Fanuc TP program (LS listing): op5_xl_master.ls

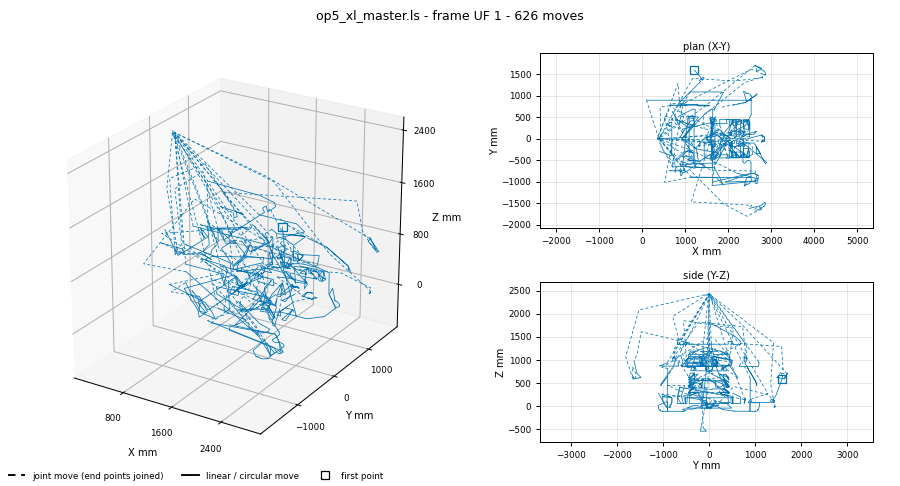
[picture p0: tool path of op5_xl_master.ls in frame UF 1, 626 of 638 moves have a stored position in this frame; points joined in program order, loops and branches not executed]
/PROG  OP5_XL_MASTER
/ATTR
OWNER		= SHIFT;
COMMENT		= "XL Main Prog";
PROG_SIZE	= 81377;
CREATE		= DATE 25-11-17  TIME 10:12:48;
MODIFIED	= DATE 26-02-12  TIME 09:04:14;
FILE_NAME	= OP5_XL_M;
VERSION		= 0;
LINE_COUNT	= 1858;
MEMORY_SIZE	= 81929;
PROTECT		= READ_WRITE;
TCD:  STACK_SIZE	= 0,
      TASK_PRIORITY	= 50,
      TIME_SLICE	= 0,
      BUSY_LAMP_OFF	= 0,
      ABORT_REQUEST	= 0,
      PAUSE_REQUEST	= 0;
DEFAULT_GROUP	= 1,1,*,*,*;
CONTROL_CODE	= 00000000 00000000;
/APPL
  ARC Welding Equipment : 1,*,*,*,*;

MPAS ;
MPAS_NUM_PASSES        : 0;
MPAS_LAST_PASS         : 0;
MPAS_CURRENT_PASS      : 0;
MPAS_STATUS_PASS       : 0;
/MN
   1:  !********** WAR HAMMER ********** ;
   2:  !-           FRAME XL           - ;
   3:  !******** FR500 CELL: C ********* ;
   4:   ;
   5:  CALL HOME    ;
   6:  CALL LOAD_POS    ;
   7:  UFRAME_NUM[GP2]=0 ;
   8:   ;
   9:  !********POSITIONER MOVE******** ;
  10:J P[1] 60% FINE    ;
  11:   ;
  12:L P[2] 1000mm/sec CNT25    ;
  13:   ;
  14:  !FR50X1000 ;
  15:  IF R[15]=1003,CALL TECH_HOLD ;
  16:   ;
  17:L P[3] 800mm/sec FINE
    :  Arc Start[6]    ;
  18:  Weave Sine[6] ;
  19:  Track TAST[6] ;
  20:L P[4] WELD_SPEED FINE
    :  Arc End[6]    ;
  21:  Weave End ;
  22:  Track End ;
  23:   ;
  24:L P[5] 1000mm/sec CNT50    ;
  25:   ;
  26:L P[6] 1000mm/sec CNT50    ;
  27:   ;
  28:   ;
  29:  !FR50X1010 ;
  30:  IF R[15]=1013,CALL TECH_HOLD ;
  31:   ;
  32:L P[7] 800mm/sec FINE
    :  Arc Start[6]    ;
  33:  Weave Sine[6] ;
  34:  Track TAST[6] ;
  35:L P[8] WELD_SPEED FINE
    :  Arc End[6]    ;
  36:  Weave End ;
  37:  Track End ;
  38:   ;
  39:L P[9] 1000mm/sec CNT25    ;
  40:   ;
  41:  !FR50X1020 ;
  42:  IF R[15]=1023,CALL TECH_HOLD ;
  43:   ;
  44:L P[10] 800mm/sec FINE
    :  Arc Start[6]    ;
  45:  Weave Sine[6] ;
  46:  Track TAST[6] ;
  47:L P[11] WELD_SPEED CNT100    ;
  48:L P[12] WELD_SPEED FINE
    :  Arc End[6]    ;
  49:  Weave End ;
  50:  Track End ;
  51:   ;
  52:L P[13] 1000mm/sec CNT25    ;
  53:   ;
  54:J P[14] 50% CNT25    ;
  55:   ;
  56:  !HOME ;
  57:J P[15] 75% CNT25    ;
  58:   ;
  59:  !********POSITIONER MOVE******** ;
  60:J P[16] 75% FINE    ;
  61:   ;
  62:J P[17] 50% CNT100    ;
  63:   ;
  64:J P[18] 50% CNT25    ;
  65:   ;
  66:  !FR50X1030 ;
  67:  IF R[15]=1033,CALL TECH_HOLD ;
  68:   ;
  69:L P[19] 800mm/sec FINE
    :  Arc Start[6]    ;
  70:  Weave Sine[6] ;
  71:  Track TAST[6] ;
  72:L P[20] WELD_SPEED FINE
    :  Arc End[6]    ;
  73:  Weave End ;
  74:  Track End ;
  75:   ;
  76:L P[21] 1000mm/sec CNT25    ;
  77:   ;
  78:J P[22] 50% CNT25    ;
  79:   ;
  80:L P[23] 1000mm/sec CNT25    ;
  81:   ;
  82:  !FR50X1040 ;
  83:  IF R[15]=1043,CALL TECH_HOLD ;
  84:   ;
  85:L P[24] 800mm/sec FINE
    :  Arc Start[6]    ;
  86:  Weave Sine[6] ;
  87:  Track TAST[6] ;
  88:L P[25] WELD_SPEED FINE
    :  Arc End[6]    ;
  89:  Weave End ;
  90:  Track End ;
  91:   ;
  92:L P[26] 960mm/sec CNT25    ;
  93:   ;
  94:J P[27] 50% CNT25    ;
  95:   ;
  96:   ;
  97:L P[28] 1000mm/sec CNT25    ;
  98:   ;
  99:  !FR50X1050 ;
 100:  IF R[15]=1053,CALL TECH_HOLD ;
 101:   ;
 102:L P[29] 800mm/sec FINE
    :  Arc Start[6]    ;
 103:  Weave Sine[6] ;
 104:  Track TAST[6] ;
 105:L P[30] WELD_SPEED CNT100    ;
 106:L P[31] WELD_SPEED FINE
    :  Arc End[6]    ;
 107:  Weave End ;
 108:  Track End ;
 109:   ;
 110:L P[32] 960mm/sec CNT25    ;
 111:   ;
 112:J P[33] 50% CNT25    ;
 113:   ;
 114:L P[34] 1000mm/sec CNT25    ;
 115:   ;
 116:  !FR50X1060 ;
 117:  IF R[15]=1063,CALL TECH_HOLD ;
 118:   ;
 119:L P[35] 800mm/sec FINE
    :  Arc Start[6]    ;
 120:  Weave Sine[6] ;
 121:  Track TAST[6] ;
 122:L P[36] WELD_SPEED CNT100    ;
 123:L P[37] WELD_SPEED FINE
    :  Arc End[6]    ;
 124:  Weave End ;
 125:  Track End ;
 126:   ;
 127:L P[38] 1000mm/sec CNT25    ;
 128:   ;
 129:J P[39] 50% CNT25    ;
 130:   ;
 131:L P[40] 1000mm/sec CNT25    ;
 132:   ;
 133:  !FR50X1070 ;
 134:  IF R[15]=1073,CALL TECH_HOLD ;
 135:   ;
 136:L P[41] 500mm/sec FINE
    :  Arc Start[6]    ;
 137:  Weave Sine[6] ;
 138:  Track TAST[6] ;
 139:L P[42] WELD_SPEED CNT100    ;
 140:L P[43] WELD_SPEED CNT100    ;
 141:L P[44] WELD_SPEED FINE
    :  Arc End[6]    ;
 142:  Weave End ;
 143:  Track End ;
 144:   ;
 145:L P[45] 700mm/sec CNT25    ;
 146:   ;
 147:L P[46] 1000mm/sec CNT50    ;
 148:   ;
 149:  !FR50X1080 ;
 150:  IF R[15]=1083,CALL TECH_HOLD ;
 151:   ;
 152:L P[47] 800mm/sec FINE
    :  Arc Start[6]    ;
 153:  Weave Sine[6] ;
 154:  Track TAST[6] ;
 155:L P[48] WELD_SPEED FINE
    :  Arc End[6]    ;
 156:  Weave End ;
 157:  Track End ;
 158:   ;
 159:L P[49] 1000mm/sec CNT25    ;
 160:   ;
 161:L P[50] 960mm/sec CNT25    ;
 162:   ;
 163:J P[51] 50% CNT25    ;
 164:   ;
 165:L P[52] 1000mm/sec CNT25    ;
 166:   ;
 167:  !FR50X1090 ;
 168:  IF R[15]=1093,CALL TECH_HOLD ;
 169:   ;
 170:L P[53] 800mm/sec FINE
    :  Arc Start[6]    ;
 171:  Weave Sine[6] ;
 172:  Track TAST[6] ;
 173:L P[54] WELD_SPEED CNT100    ;
 174:L P[55] WELD_SPEED CNT100    ;
 175:L P[56] WELD_SPEED FINE
    :  Arc End[6]    ;
 176:  Weave End ;
 177:  Track End ;
 178:   ;
 179:L P[57] 1000mm/sec CNT25    ;
 180:   ;
 181:L P[58] 1000mm/sec CNT50    ;
 182:   ;
 183:  !FR50X1100 ;
 184:  IF R[15]=1103,CALL TECH_HOLD ;
 185:   ;
 186:L P[59] 800mm/sec FINE
    :  Arc Start[6]    ;
 187:  Weave Sine[6] ;
 188:  Track TAST[6] ;
 189:L P[60] WELD_SPEED FINE
    :  Arc End[6]    ;
 190:  Weave End ;
 191:  Track End ;
 192:   ;
 193:L P[61] 1000mm/sec CNT25    ;
 194:   ;
 195:J P[62] 50% CNT25    ;
 196:   ;
 197:L P[63] 1000mm/sec CNT25    ;
 198:   ;
 199:  !FR50X1110 ;
 200:  IF R[15]=1113,CALL TECH_HOLD ;
 201:   ;
 202:L P[64] 800mm/sec FINE
    :  Arc Start[8]    ;
 203:  Weave Sine[8] ;
 204:L P[65] WELD_SPEED CNT100    ;
 205:L P[66] WELD_SPEED FINE
    :  Arc End[8]    ;
 206:  Weave End ;
 207:   ;
 208:L P[67] 800mm/sec CNT25    ;
 209:   ;
 210:J P[68] 50% CNT25    ;
 211:   ;
 212:  !********POSITIONER MOVE******** ;
 213:J P[69] 75% FINE    ;
 214:   ;
 215:  !FR50X1120 ;
 216:  IF R[15]=1123,CALL TECH_HOLD ;
 217:   ;
 218:L P[70] 800mm/sec FINE
    :  Arc Start[8]    ;
 219:  Weave Sine[8] ;
 220:L P[71] WELD_SPEED FINE
    :  Arc End[8]    ;
 221:  Weave End ;
 222:   ;
 223:L P[72] 1000mm/sec CNT25    ;
 224:   ;
 225:J P[73] 50% CNT25    ;
 226:   ;
 227:  !HOME ;
 228:J P[74] 100% FINE    ;
 229:   ;
 230:  !********POSITIONER MOVE******** ;
 231:J P[75] 60% FINE    ;
 232:   ;
 233:J P[76] 50% CNT25    ;
 234:   ;
 235:L P[77] 1000mm/sec CNT25    ;
 236:   ;
 237:L P[78] 500mm/sec CNT25    ;
 238:   ;
 239:  !FR50X1130 ;
 240:  IF R[15]=1133,CALL TECH_HOLD ;
 241:   ;
 242:L P[79] 400mm/sec FINE
    :  Arc Start[6]    ;
 243:  Weave Sine[6] ;
 244:L P[80] WELD_SPEED FINE
    :  Arc End[6]    ;
 245:  Weave End ;
 246:   ;
 247:L P[81] 500mm/sec CNT25    ;
 248:   ;
 249:L P[82] 1000mm/sec CNT25    ;
 250:   ;
 251:J P[83] 40% CNT25    ;
 252:   ;
 253:J P[84] 50% CNT25    ;
 254:   ;
 255:  !HOME ;
 256:J P[85] 100% FINE    ;
 257:   ;
 258:  !********POSITIONER MOVE******** ;
 259:J P[86] 70% FINE    ;
 260:   ;
 261:J P[87] 50% CNT25    ;
 262:   ;
 263:L P[88] 1000mm/sec CNT25    ;
 264:   ;
 265:L P[89] 1000mm/sec CNT25    ;
 266:   ;
 267:  !FR50X1140 ;
 268:  IF R[15]=1143,CALL TECH_HOLD ;
 269:   ;
 270:L P[90] 700mm/sec FINE
    :  Arc Start[6]    ;
 271:  Weave Sine[6] ;
 272:  Track TAST[6] ;
 273:L P[91] WELD_SPEED CNT100    ;
 274:L P[92] WELD_SPEED FINE
    :  Arc End[6]    ;
 275:  Weave End ;
 276:  Track End ;
 277:   ;
 278:L P[93] 1000mm/sec CNT25    ;
 279:   ;
 280:L P[94] 1000mm/sec CNT25    ;
 281:   ;
 282:L P[95] 1000mm/sec CNT25    ;
 283:   ;
 284:J P[96] 50% CNT25    ;
 285:   ;
 286:L P[97] 1000mm/sec CNT25    ;
 287:   ;
 288:  !FR50X1150 ;
 289:  IF R[15]=1153,CALL TECH_HOLD ;
 290:   ;
 291:L P[98] 1000mm/sec FINE
    :  Arc Start[6]    ;
 292:  Weave Sine[6] ;
 293:  Track TAST[6] ;
 294:L P[99] WELD_SPEED CNT100    ;
 295:L P[100] WELD_SPEED FINE
    :  Arc End[6]    ;
 296:  Weave End ;
 297:  Track End ;
 298:   ;
 299:L P[101] 1000mm/sec CNT25    ;
 300:   ;
 301:L P[102] 1000mm/sec CNT25    ;
 302:   ;
 303:  !********POSITIONER MOVE******** ;
 304:J P[103] 75% FINE    ;
 305:   ;
 306:L P[104] 1000mm/sec CNT25    ;
 307:   ;
 308:L P[105] 1000mm/sec CNT25    ;
 309:   ;
 310:  !FR50X1160 ;
 311:  IF R[15]=1163,CALL TECH_HOLD ;
 312:   ;
 313:L P[106] 1000mm/sec FINE
    :  Arc Start[6]    ;
 314:  Weave Sine[6] ;
 315:  Track TAST[6] ;
 316:L P[107] WELD_SPEED FINE
    :  Arc End[6]    ;
 317:  Weave End ;
 318:  Track End ;
 319:   ;
 320:L P[108] 1000mm/sec CNT25    ;
 321:   ;
 322:  !FR50X1170 ;
 323:  IF R[15]=1173,CALL TECH_HOLD ;
 324:   ;
 325:L P[109] 1000mm/sec FINE
    :  Arc Start[6]    ;
 326:  Weave Sine[6] ;
 327:  Track TAST[6] ;
 328:L P[110] WELD_SPEED FINE
    :  Arc End[6]    ;
 329:  Weave End ;
 330:  Track End ;
 331:   ;
 332:L P[111] 1000mm/sec CNT25    ;
 333:   ;
 334:L P[112] 1000mm/sec CNT25    ;
 335:   ;
 336:  !FR50X1180 ;
 337:  IF R[15]=1183,CALL TECH_HOLD ;
 338:   ;
 339:L P[113] 1000mm/sec FINE
    :  Arc Start[6]    ;
 340:  Weave Sine[6] ;
 341:  Track TAST[6] ;
 342:L P[114] WELD_SPEED FINE
    :  Arc End[6]    ;
 343:  Weave End ;
 344:  Track End ;
 345:   ;
 346:L P[115] 1000mm/sec CNT25    ;
 347:   ;
 348:L P[116] 1000mm/sec CNT25    ;
 349:   ;
 350:  !FR50X1190 ;
 351:  IF R[15]=1193,CALL TECH_HOLD ;
 352:   ;
 353:L P[117] 1000mm/sec FINE
    :  Arc Start[6]    ;
 354:  Weave Sine[6] ;
 355:  Track TAST[6] ;
 356:L P[118] WELD_SPEED FINE
    :  Arc End[6]    ;
 357:  Weave End ;
 358:  Track End ;
 359:   ;
 360:L P[119] 1000mm/sec CNT25    ;
 361:   ;
 362:L P[120] 1000mm/sec CNT25    ;
 363:   ;
 364:  !FR50X1200 ;
 365:  IF R[15]=1203,CALL TECH_HOLD ;
 366:   ;
 367:L P[121] 1000mm/sec FINE
    :  Arc Start[6]    ;
 368:  Weave Sine[6] ;
 369:  Track TAST[6] ;
 370:L P[122] WELD_SPEED FINE
    :  Arc End[6]    ;
 371:  Weave End ;
 372:  Track End ;
 373:   ;
 374:L P[123] 1000mm/sec CNT25    ;
 375:   ;
 376:L P[124] 1000mm/sec CNT25    ;
 377:   ;
 378:J P[125] 50% CNT25    ;
 379:   ;
 380:  !********POSITIONER MOVE******** ;
 381:J P[126] 75% FINE    ;
 382:   ;
 383:L P[127] 1000mm/sec CNT25    ;
 384:   ;
 385:  !FR50X1210 ;
 386:  IF R[15]=1213,CALL TECH_HOLD ;
 387:   ;
 388:L P[128] 500mm/sec FINE
    :  Arc Start[6]    ;
 389:  Weave Sine[6] ;
 390:  Track TAST[6] ;
 391:L P[129] WELD_SPEED FINE
    :  Arc End[6]    ;
 392:  Weave End ;
 393:  Track End ;
 394:   ;
 395:L P[130] 500mm/sec CNT25    ;
 396:   ;
 397:L P[131] 1000mm/sec FINE    ;
 398:   ;
 399:J P[132] 50% CNT25    ;
 400:   ;
 401:  !********POSITIONER MOVE******** ;
 402:J P[133] 75% FINE    ;
 403:   ;
 404:J P[134] 50% CNT25    ;
 405:   ;
 406:L P[135] 1000mm/sec CNT25    ;
 407:   ;
 408:  !FR50X1220 ;
 409:  IF R[15]=1223,CALL TECH_HOLD ;
 410:   ;
 411:L P[136] 1000mm/sec FINE
    :  Arc Start[6]    ;
 412:  Weave Sine[6] ;
 413:  Track TAST[6] ;
 414:L P[137] WELD_SPEED FINE
    :  Arc End[6]    ;
 415:  Weave End ;
 416:  Track End ;
 417:   ;
 418:L P[138] 500mm/sec CNT25    ;
 419:   ;
 420:J P[139] 50% CNT25    ;
 421:   ;
 422:J P[140] 50% CNT25    ;
 423:   ;
 424:  !HOME ;
 425:J P[141] 100% FINE    ;
 426:   ;
 427:  !********POSITIONER MOVE******** ;
 428:J P[142] 75% FINE    ;
 429:   ;
 430:  !TORCH CLEAN ;
 431:  CALL T_CLEAN    ;
 432:   ;
 433:   ;
 434:J P[143] 50% CNT25    ;
 435:   ;
 436:L P[144] 960mm/sec CNT25    ;
 437:   ;
 438:  !FR50X1230 ;
 439:  IF R[15]=1233,CALL TECH_HOLD ;
 440:   ;
 441:L P[145] 800mm/sec FINE
    :  Arc Start[6]    ;
 442:  Weave Sine[6] ;
 443:  Track TAST[6] ;
 444:L P[146] WELD_SPEED FINE
    :  Arc End[6]    ;
 445:  Weave End ;
 446:  Track End ;
 447:   ;
 448:L P[147] 960mm/sec CNT25    ;
 449:   ;
 450:J P[148] 50% CNT25    ;
 451:   ;
 452:  !FR50X1240 ;
 453:  IF R[15]=1243,CALL TECH_HOLD ;
 454:   ;
 455:L P[149] 800mm/sec FINE
    :  Arc Start[3]    ;
 456:L P[150] WELD_SPEED CNT100    ;
 457:L P[151] WELD_SPEED FINE
    :  Arc End[3]    ;
 458:   ;
 459:L P[152] 1000mm/sec CNT25    ;
 460:   ;
 461:L P[153] 500mm/sec CNT25    ;
 462:   ;
 463:  //UALM[20] ;
 464:   ;
 465:  !FR50X1250 ;
 466:  IF R[15]=1253,CALL TECH_HOLD ;
 467:   ;
 468:L P[154] 800mm/sec FINE
    :  Arc Start[3]    ;
 469:L P[155] WELD_SPEED CNT100    ;
 470:L P[156] WELD_SPEED FINE
    :  Arc End[3]    ;
 471:   ;
 472:L P[157] 1000mm/sec CNT25    ;
 473:   ;
 474:J P[158] 50% CNT25    ;
 475:   ;
 476:L P[159] 1000mm/sec CNT25    ;
 477:   ;
 478:  !FR50X1260 ;
 479:  IF R[15]=1263,CALL TECH_HOLD ;
 480:   ;
 481:L P[160] 800mm/sec FINE
    :  Arc Start[6]    ;
 482:  Weave Sine[6] ;
 483:  Track TAST[6] ;
 484:L P[161] WELD_SPEED FINE
    :  Arc End[6]    ;
 485:  Track End ;
 486:  Weave End ;
 487:   ;
 488:L P[162] 1000mm/sec CNT25    ;
 489:   ;
 490:L P[163] 1000mm/sec CNT25    ;
 491:   ;
 492:L P[164] 1000mm/sec CNT25    ;
 493:   ;
 494:  !FR50X1270 ;
 495:  IF R[15]=1273,CALL TECH_HOLD ;
 496:   ;
 497:L P[165] 800mm/sec FINE
    :  Arc Start[6]    ;
 498:  Weave Sine[6] ;
 499:  Track TAST[6] ;
 500:L P[166] WELD_SPEED FINE
    :  Arc End[6]    ;
 501:  Weave End ;
 502:  Track End ;
 503:   ;
 504:L P[167] 1000mm/sec CNT25    ;
 505:   ;
 506:J P[168] 50% CNT25    ;
 507:   ;
 508:  !********POSITIONER MOVE******** ;
 509:J P[169] 75% FINE    ;
 510:   ;
 511:L P[170] 1000mm/sec CNT25    ;
 512:   ;
 513:  !FR50X1280 ;
 514:  IF R[15]=1283,CALL TECH_HOLD ;
 515:   ;
 516:L P[171] 1000mm/sec FINE
    :  Arc Start[6]    ;
 517:  Weave Sine[6] ;
 518:  Track TAST[6] ;
 519:L P[172] WELD_SPEED FINE
    :  Arc End[6]    ;
 520:  Weave End ;
 521:  Track End ;
 522:   ;
 523:L P[173] 500mm/sec CNT25    ;
 524:   ;
 525:L P[174] 1000mm/sec CNT25    ;
 526:   ;
 527:L P[175] 1000mm/sec FINE    ;
 528:   ;
 529:  !********POSITIONER MOVE******** ;
 530:J P[176] 75% FINE    ;
 531:   ;
 532:L P[177] 1000mm/sec CNT25    ;
 533:   ;
 534:  !FR50X1290 ;
 535:  IF R[15]=1293,CALL TECH_HOLD ;
 536:   ;
 537:L P[178] 800mm/sec FINE
    :  Arc Start[6]    ;
 538:  Weave Sine[6] ;
 539:  Track TAST[6] ;
 540:L P[179] WELD_SPEED FINE
    :  Arc End[6]    ;
 541:  Weave End ;
 542:  Track End ;
 543:   ;
 544:L P[180] 300mm/sec FINE    ;
 545:   ;
 546:L P[181] 1000mm/sec FINE    ;
 547:   ;
 548:J P[182] 50% CNT25    ;
 549:   ;
 550:  !HOME ;
 551:J P[183] 100% FINE    ;
 552:   ;
 553:  !********POSITIONER MOVE******** ;
 554:J P[184] 75% FINE    ;
 555:   ;
 556:J P[185] 50% CNT25    ;
 557:   ;
 558:   ;
 559:  !FR50X1300 ;
 560:  IF R[15]=1303,CALL TECH_HOLD ;
 561:   ;
 562:   ;
 563:L P[186] 800mm/sec FINE
    :  Arc Start[6]    ;
 564:  Weave Sine[6] ;
 565:  Track TAST[6] ;
 566:L P[187] WELD_SPEED FINE
    :  Arc End[6]    ;
 567:  Weave End ;
 568:  Track End ;
 569:   ;
 570:L P[188] 1000mm/sec CNT25    ;
 571:   ;
 572:L P[189] 1000mm/sec CNT30    ;
 573:   ;
 574:  !FR50X1310 ;
 575:  IF R[15]=1313,CALL TECH_HOLD ;
 576:   ;
 577:L P[190] 800mm/sec FINE
    :  Arc Start[6]    ;
 578:  Weave Sine[6] ;
 579:  Track TAST[6] ;
 580:L P[191] WELD_SPEED FINE
    :  Arc End[6]    ;
 581:  Weave End ;
 582:  Track End ;
 583:   ;
 584:L P[192] 1000mm/sec CNT25    ;
 585:   ;
 586:  !FR50X1320 ;
 587:  IF R[15]=1323,CALL TECH_HOLD ;
 588:   ;
 589:L P[194] 800mm/sec FINE
    :  Arc Start[6]    ;
 590:  Weave Sine[6] ;
 591:  Track TAST[6] ;
 592:L P[195] WELD_SPEED FINE
    :  Arc End[6]    ;
 593:  Weave End ;
 594:  Track End ;
 595:   ;
 596:L P[196] 1000mm/sec CNT25    ;
 597:   ;
 598:  !********POSITIONER MOVE******** ;
 599:J P[197] 100% CNT25    ;
 600:   ;
 601:L P[198] 1000mm/sec CNT25    ;
 602:   ;
 603:  CALL ARC_DISABLE_RH_LS(0) ;
 604:   ;
 605:  //UALM[20] ;
 606:   ;
 607:  !FR50X1330 ;
 608:  IF R[15]=1333,CALL TECH_HOLD ;
 609:   ;
 610:L P[199] 800mm/sec FINE
    :  Arc Start[8]    ;
 611:  Weave Sine[8] ;
 612:L P[200] WELD_SPEED FINE
    :  Arc End[8]    ;
 613:  Weave End ;
 614:   ;
 615:L P[201] 800mm/sec FINE    ;
 616:   ;
 617:L P[202] 1000mm/sec CNT25    ;
 618:   ;
 619:J P[203] 50% CNT25    ;
 620:   ;
 621:  !FR50X1340 ;
 622:  !LENGTH: 57mm ;
 623:  IF R[15]=1343,CALL TECH_HOLD ;
 624:   ;
 625:L P[204] 800mm/sec FINE
    :  Arc Start[8]    ;
 626:  Weave Sine[8] ;
 627:L P[205] WELD_SPEED FINE
    :  Arc End[8]    ;
 628:  Weave End ;
 629:   ;
 630:  CALL ARC_DISABLE_RH_LS(1) ;
 631:   ;
 632:L P[206] 800mm/sec CNT5    ;
 633:   ;
 634:  !********POSITIONER MOVE******** ;
 635:J P[207] 50% CNT25    ;
 636:   ;
 637:J P[208] 50% CNT25    ;
 638:   ;
 639:J P[209] 25% CNT25    ;
 640:   ;
 641:  DO[89:OFF:Inch backward   ]=PULSE,0.8sec ;
 642:   ;
 643:  CALL ARC_LH_DISABLE_LS(0) ;
 644:   ;
 645:  !FR50X1350 ;
 646:  IF R[15]=1353,CALL TECH_HOLD ;
 647:   ;
 648:L P[210] 500mm/sec FINE
    :  Arc Start[8]    ;
 649:  Weave Sine[8] ;
 650:L P[211] WELD_SPEED FINE
    :  Arc End[8]    ;
 651:  Weave End ;
 652:   ;
 653:L P[212] 100mm/sec CNT5    ;
 654:   ;
 655:L P[213] 1000mm/sec CNT25    ;
 656:   ;
 657:J P[214] 100% CNT25    ;
 658:   ;
 659:  !FR50X1360 ;
 660:  !LENGTH: 57mm ;
 661:  IF R[15]=1363,CALL TECH_HOLD ;
 662:   ;
 663:L P[215] 800mm/sec FINE
    :  Arc Start[8]    ;
 664:  Weave Sine[8] ;
 665:L P[216] WELD_SPEED FINE
    :  Arc End[8]    ;
 666:  Weave End ;
 667:   ;
 668:  CALL ARC_LH_DISABLE_LS(1) ;
 669:   ;
 670:L P[217] 100mm/sec CNT25    ;
 671:   ;
 672:J P[218] 100% CNT25    ;
 673:   ;
 674:  !HOME ;
 675:J P[219] 100% FINE    ;
 676:   ;
 677:  !********POSITIONER MOVE******** ;
 678:J P[220] 75% FINE    ;
 679:   ;
 680:J P[221] 50% CNT25    ;
 681:   ;
 682:J P[222] 50% CNT25    ;
 683:   ;
 684:   ;
 685:L P[193] 1000mm/sec CNT25    ;
 686:   ;
 687:  !FR50X1370 ;
 688:  IF R[15]=1373,CALL TECH_HOLD ;
 689:   ;
 690:L P[672] 800mm/sec FINE
    :  Arc Start[6]    ;
 691:  Weave Sine[6] ;
 692:L P[673] WELD_SPEED FINE
    :  Arc End[6]    ;
 693:  Weave End ;
 694:   ;
 695:L P[674] 1000mm/sec CNT25    ;
 696:   ;
 697:J P[675] 50% CNT25    ;
 698:   ;
 699:L P[676] 800mm/sec CNT10    ;
 700:   ;
 701:  !FR50X1380 ;
 702:  IF R[15]=1383,CALL TECH_HOLD ;
 703:   ;
 704:L P[677] 800mm/sec FINE
    :  Arc Start[6]    ;
 705:  Weave Sine[6] ;
 706:L P[678] WELD_SPEED FINE
    :  Arc End[6]    ;
 707:  Weave End ;
 708:   ;
 709:L P[679] 1000mm/sec CNT25    ;
 710:   ;
 711:J P[680] 50% CNT25    ;
 712:   ;
 713:L P[681] 500mm/sec CNT25    ;
 714:   ;
 715:  !FR50X1390 ;
 716:  IF R[15]=1393,CALL TECH_HOLD ;
 717:   ;
 718:L P[682] 800mm/sec FINE
    :  Arc Start[6]    ;
 719:  Weave Sine[6] ;
 720:L P[683] WELD_SPEED FINE
    :  Arc End[6]    ;
 721:  Weave End ;
 722:   ;
 723:L P[684] 500mm/sec CNT25    ;
 724:   ;
 725:J P[685] 50% CNT25    ;
 726:   ;
 727:J P[686] 50% CNT25    ;
 728:   ;
 729:J P[687] 50% CNT30    ;
 730:   ;
 731:   ;
 732:   ;
 733:  !FR50X1400 ;
 734:  IF R[15]=1403,CALL TECH_HOLD ;
 735:   ;
 736:L P[688] 800mm/sec FINE
    :  Arc Start[6]    ;
 737:  Weave Sine[6] ;
 738:  Track TAST[6] ;
 739:L P[689] WELD_SPEED FINE
    :  Arc End[6]    ;
 740:  Weave End ;
 741:  Track End ;
 742:   ;
 743:L P[690] 1000mm/sec CNT25    ;
 744:   ;
 745:L P[691] 1000mm/sec CNT25    ;
 746:   ;
 747:  !FR50X1410 ;
 748:  IF R[15]=1413,CALL TECH_HOLD ;
 749:   ;
 750:L P[692] 800mm/sec FINE
    :  Arc Start[6]    ;
 751:  Weave Sine[6] ;
 752:  Track TAST[6] ;
 753:L P[693] WELD_SPEED FINE
    :  Arc End[6]    ;
 754:  Weave End ;
 755:  Track End ;
 756:   ;
 757:L P[694] 1000mm/sec CNT25    ;
 758:   ;
 759:J P[695] 50% CNT25    ;
 760:   ;
 761:   ;
 762:  !FR50X1420 ;
 763:  IF R[15]=1423,CALL TECH_HOLD ;
 764:   ;
 765:L P[696] 800mm/sec FINE
    :  Arc Start[6]    ;
 766:  Weave Sine[6] ;
 767:  Track TAST[6] ;
 768:L P[697] WELD_SPEED CNT100    ;
 769:C P[698]
    :  P[699] WELD_SPEED FINE
    :  Arc End[6]    ;
 770:  Weave End ;
 771:  Track End ;
 772:   ;
 773:L P[700] 1000mm/sec CNT25    ;
 774:   ;
 775:J P[701] 50% CNT25    ;
 776:   ;
 777:J P[702] 50% CNT25    ;
 778:   ;
 779:   ;
 780:   ;
 781:  !FR50X1430 ;
 782:  IF R[15]=1433,CALL TECH_HOLD ;
 783:   ;
 784:L P[703] 800mm/sec FINE
    :  Arc Start[6]    ;
 785:  Weave Sine[6] ;
 786:  Track TAST[6] ;
 787:L P[704] WELD_SPEED FINE
    :  Arc End[6]    ;
 788:  Track End ;
 789:  Weave End ;
 790:   ;
 791:L P[705] 1000mm/sec CNT25    ;
 792:   ;
 793:L P[706] 1000mm/sec CNT25    ;
 794:   ;
 795:  !FR50X1440 ;
 796:  IF R[15]=1443,CALL TECH_HOLD ;
 797:   ;
 798:L P[707] 800mm/sec FINE
    :  Arc Start[6]    ;
 799:  Weave Sine[6] ;
 800:  Track TAST[6] ;
 801:L P[708] WELD_SPEED FINE
    :  Arc End[6]    ;
 802:  Weave End ;
 803:  Track End ;
 804:   ;
 805:L P[709] 1000mm/sec CNT25    ;
 806:   ;
 807:J P[710] 50% CNT25    ;
 808:   ;
 809:  //UALM[20] ;
 810:  //--eg:TOUCH UP ;
 811:   ;
 812:  !FR50X1450 ;
 813:  IF R[15]=1453,CALL TECH_HOLD ;
 814:   ;
 815:L P[711] 800mm/sec FINE
    :  Arc Start[6]    ;
 816:  Weave Sine[6] ;
 817:  Track TAST[6] ;
 818:L P[712] WELD_SPEED CNT100    ;
 819:C P[713]
    :  P[714] WELD_SPEED FINE
    :  Arc End[6]    ;
 820:  Weave End ;
 821:  Track End ;
 822:   ;
 823:L P[715] 960mm/sec FINE    ;
 824:   ;
 825:J P[716] 50% CNT25    ;
 826:   ;
 827:L P[717] 1000mm/sec CNT25    ;
 828:   ;
 829:  !FR50X1460 ;
 830:  IF R[15]=1463,CALL TECH_HOLD ;
 831:   ;
 832:L P[718] 800mm/sec FINE
    :  Arc Start[6]    ;
 833:  Weave Sine[6] ;
 834:  Track TAST[6] ;
 835:L P[719] WELD_SPEED FINE
    :  Arc End[6]    ;
 836:  Weave End ;
 837:  Track End ;
 838:   ;
 839:L P[720] 1000mm/sec CNT25    ;
 840:   ;
 841:L P[721] 1000mm/sec CNT25    ;
 842:   ;
 843:L P[722] 1000mm/sec CNT25    ;
 844:   ;
 845:L P[723] 1000mm/sec CNT25    ;
 846:   ;
 847:  !FR50X1470 ;
 848:  IF R[15]=1473,CALL TECH_HOLD ;
 849:   ;
 850:L P[724] 200mm/sec FINE
    :  Arc Start[6]    ;
 851:  Weave Sine[6] ;
 852:  Track TAST[6] ;
 853:L P[725] WELD_SPEED FINE
    :  Arc End[6]    ;
 854:  Weave End ;
 855:  Track End ;
 856:   ;
 857:L P[726] 200mm/sec CNT25    ;
 858:   ;
 859:L P[727] 1000mm/sec FINE    ;
 860:   ;
 861:J P[728] 50% FINE    ;
 862:   ;
 863:L P[729] 1000mm/sec CNT25    ;
 864:   ;
 865:  !FR50X1480 ;
 866:  IF R[15]=1483,CALL TECH_HOLD ;
 867:   ;
 868:L P[730] 800mm/sec FINE
    :  Arc Start[6]    ;
 869:  Weave Sine[6] ;
 870:  Track TAST[6] ;
 871:L P[731] WELD_SPEED FINE
    :  Arc End[6]    ;
 872:  Weave End ;
 873:  Track End ;
 874:   ;
 875:L P[732] 1000mm/sec CNT25    ;
 876:   ;
 877:L P[733] 500mm/sec CNT25    ;
 878:   ;
 879:L P[734] 500mm/sec CNT25    ;
 880:   ;
 881:  !FR50X1490 ;
 882:  IF R[15]=1493,CALL TECH_HOLD ;
 883:   ;
 884:L P[735] 300mm/sec FINE
    :  Arc Start[6]    ;
 885:  Weave Sine[6] ;
 886:  Track TAST[6] ;
 887:L P[736] WELD_SPEED FINE
    :  Arc End[6]    ;
 888:  Weave End ;
 889:  Track End ;
 890:   ;
 891:L P[737] 300mm/sec CNT25    ;
 892:   ;
 893:J P[738] 25% FINE    ;
 894:   ;
 895:L P[739] 1000mm/sec CNT25    ;
 896:   ;
 897:  !HOME ;
 898:J P[740] 100% FINE    ;
 899:   ;
 900:  !********POSITIONER MOVE******** ;
 901:J P[741] 75% FINE    ;
 902:   ;
 903:J P[742] 50% CNT40    ;
 904:   ;
 905:L P[743] 1000mm/sec CNT25    ;
 906:   ;
 907:  !FR50X1500 ;
 908:  !LENGTH: 100mm ;
 909:  IF R[15]=1503,CALL TECH_HOLD ;
 910:   ;
 911:L P[744] 800mm/sec FINE
    :  Arc Start[8]    ;
 912:  Weave Sine[8] ;
 913:L P[745] WELD_SPEED FINE
    :  Arc End[8]    ;
 914:  Weave End ;
 915:   ;
 916:L P[746] 1000mm/sec CNT25    ;
 917:   ;
 918:  !FR50X1510 ;
 919:  !LENGTH: 85mm ;
 920:  IF R[15]=1513,CALL TECH_HOLD ;
 921:   ;
 922:L P[747] 800mm/sec FINE
    :  Arc Start[8]    ;
 923:  Weave Sine[8] ;
 924:L P[748] WELD_SPEED FINE
    :  Arc End[8]    ;
 925:  Weave End ;
 926:   ;
 927:L P[749] 1000mm/sec CNT25    ;
 928:   ;
 929:L P[750] 1000mm/sec CNT25    ;
 930:   ;
 931:   ;
 932:  !FR50X1520 ;
 933:  !LENGTH: 100mm - 1 of 2 ;
 934:  IF R[15]=1523,CALL TECH_HOLD ;
 935:   ;
 936:L P[751] 800mm/sec FINE
    :  Arc Start[8]    ;
 937:  Weave Sine[8] ;
 938:L P[752] WELD_SPEED FINE
    :  Arc End[8]    ;
 939:  Weave End ;
 940:   ;
 941:L P[753] 1000mm/sec CNT25    ;
 942:   ;
 943:L P[754] 1000mm/sec CNT100    ;
 944:   ;
 945:   ;
 946:   ;
 947:  !FR50X1530 ;
 948:  !LENGTH: 100mm - 2 of 2 ;
 949:  IF R[15]=1533,CALL TECH_HOLD ;
 950:   ;
 951:L P[755] 800mm/sec FINE
    :  Arc Start[6]    ;
 952:  Weave Sine[6] ;
 953:L P[756] WELD_SPEED FINE
    :  Arc End[6]    ;
 954:  Weave End ;
 955:   ;
 956:L P[757] 1000mm/sec CNT50    ;
 957:   ;
 958:L P[758] 1000mm/sec CNT25    ;
 959:   ;
 960:  !FR50X1540 ;
 961:  !LENGTH: 85mm ;
 962:  IF R[15]=1543,CALL TECH_HOLD ;
 963:   ;
 964:L P[759] 800mm/sec FINE
    :  Arc Start[8]    ;
 965:  Weave Sine[8] ;
 966:L P[760] WELD_SPEED FINE
    :  Arc End[8]    ;
 967:  Weave End ;
 968:   ;
 969:L P[761] 1000mm/sec CNT25    ;
 970:   ;
 971:L P[762] 1000mm/sec CNT25    ;
 972:   ;
 973:J P[763] 50% CNT25    ;
 974:   ;
 975:L P[764] 1000mm/sec CNT25    ;
 976:   ;
 977:  !FR50X1550 ;
 978:  IF R[15]=1553,CALL TECH_HOLD ;
 979:   ;
 980:   ;
 981:L P[765] 800mm/sec FINE
    :  Arc Start[6]    ;
 982:  Weave Sine[6] ;
 983:  Track TAST[6] ;
 984:L P[233] WELD_SPEED CNT100    ;
 985:L P[234] WELD_SPEED CNT100    ;
 986:L P[235] WELD_SPEED CNT100    ;
 987:L P[766] WELD_SPEED FINE
    :  Arc End[6]    ;
 988:  Weave End ;
 989:  Track End ;
 990:   ;
 991:L P[767] 1000mm/sec CNT25    ;
 992:   ;
 993:  !FR50X1560 ;
 994:  IF R[15]=1563,CALL TECH_HOLD ;
 995:   ;
 996:L P[768] 800mm/sec FINE
    :  Arc Start[6]    ;
 997:  Weave Sine[6] ;
 998:  Track TAST[6] ;
 999:C P[769]
    :  P[770] WELD_SPEED FINE
    :  Arc End[6]    ;
1000:  Weave End ;
1001:  Track End ;
1002:   ;
1003:L P[771] 1000mm/sec CNT25    ;
1004:   ;
1005:L P[772] 1000mm/sec CNT25    ;
1006:   ;
1007:  !FR50X1570 ;
1008:  IF R[15]=1573,CALL TECH_HOLD ;
1009:   ;
1010:L P[773] 800mm/sec FINE
    :  Arc Start[6]    ;
1011:  Weave Sine[6] ;
1012:  Track TAST[6] ;
1013:L P[774] WELD_SPEED FINE
    :  Arc End[6]    ;
1014:  Weave End ;
1015:  Track End ;
1016:   ;
1017:L P[775] 1000mm/sec CNT25    ;
1018:   ;
1019:L P[776] 1000mm/sec CNT25    ;
1020:   ;
1021:  !FR50X1580 ;
1022:  IF R[15]=1583,CALL TECH_HOLD ;
1023:   ;
1024:L P[777] 800mm/sec FINE
    :  Arc Start[6]    ;
1025:  Weave Sine[6] ;
1026:  Track TAST[6] ;
1027:L P[778] WELD_SPEED CNT100    ;
1028:L P[779] WELD_SPEED CNT100    ;
1029:L P[780] WELD_SPEED FINE
    :  Arc End[6]    ;
1030:  Weave End ;
1031:  Track End ;
1032:   ;
1033:L P[781] 1000mm/sec CNT25    ;
1034:   ;
1035:L P[782] 1000mm/sec CNT25    ;
1036:   ;
1037:  !FR50X1590 ;
1038:  IF R[15]=1593,CALL TECH_HOLD ;
1039:   ;
1040:L P[783] 800mm/sec FINE
    :  Arc Start[6]    ;
1041:  Weave Sine[6] ;
1042:  Track TAST[6] ;
1043:L P[784] WELD_SPEED FINE
    :  Arc End[6]    ;
1044:  Weave End ;
1045:  Track End ;
1046:   ;
1047:L P[785] 1000mm/sec CNT25    ;
1048:   ;
1049:J P[786] 50% CNT25    ;
1050:   ;
1051:J P[787] 50% CNT25    ;
1052:   ;
1053:  !FR50X1600 ;
1054:  IF R[15]=1603,CALL TECH_HOLD ;
1055:   ;
1056:L P[788] 800mm/sec FINE
    :  Arc Start[6]    ;
1057:  Weave Sine[6] ;
1058:  Track TAST[6] ;
1059:L P[789] WELD_SPEED FINE
    :  Arc End[6]    ;
1060:  Weave End ;
1061:  Track End ;
1062:   ;
1063:L P[790] 1000mm/sec CNT25    ;
1064:   ;
1065:  !FR50X1610 ;
1066:  IF R[15]=1613,CALL TECH_HOLD ;
1067:   ;
1068:L P[791] 800mm/sec FINE
    :  Arc Start[6]    ;
1069:  Weave Sine[6] ;
1070:  Track TAST[6] ;
1071:C P[792]
    :  P[793] WELD_SPEED FINE
    :  Arc End[6]    ;
1072:  Weave End ;
1073:  Track End ;
1074:   ;
1075:L P[794] 1000mm/sec CNT25    ;
1076:   ;
1077:L P[795] 1000mm/sec CNT25    ;
1078:   ;
1079:   ;
1080:  !FR50X1620 ;
1081:  IF R[15]=1623,CALL TECH_HOLD ;
1082:   ;
1083:L P[796] 800mm/sec FINE
    :  Arc Start[6]    ;
1084:  Weave Sine[6] ;
1085:  Track TAST[6] ;
1086:L P[797] WELD_SPEED FINE
    :  Arc End[6]    ;
1087:  Weave End ;
1088:  Track End ;
1089:   ;
1090:L P[798] 1000mm/sec CNT25    ;
1091:   ;
1092:  !FR50X1630 ;
1093:  IF R[15]=1633,CALL TECH_HOLD ;
1094:   ;
1095:L P[799] 800mm/sec FINE
    :  Arc Start[6]    ;
1096:  Weave Sine[6] ;
1097:  Track TAST[6] ;
1098:L P[800] WELD_SPEED CNT100    ;
1099:L P[801] WELD_SPEED CNT100    ;
1100:L P[802] WELD_SPEED FINE
    :  Arc End[6]    ;
1101:  Weave End ;
1102:  Track End ;
1103:   ;
1104:L P[803] 300mm/sec CNT25    ;
1105:   ;
1106:L P[804] 300mm/sec CNT25    ;
1107:   ;
1108:  !FR50X1640 ;
1109:  IF R[15]=1643,CALL TECH_HOLD ;
1110:   ;
1111:L P[805] 800mm/sec FINE
    :  Arc Start[6]    ;
1112:  Weave Sine[6] ;
1113:  Track TAST[6] ;
1114:L P[806] WELD_SPEED FINE
    :  Arc End[6]    ;
1115:  Weave End ;
1116:  Track End ;
1117:   ;
1118:L P[807] 300mm/sec CNT5    ;
1119:   ;
1120:L P[808] 300mm/sec CNT25    ;
1121:   ;
1122:J P[809] 50% CNT25    ;
1123:   ;
1124:  !HOME ;
1125:J P[810] 100% CNT25    ;
1126:   ;
1127:  !TORCH CLEAN ;
1128:  CALL HOME    ;
1129:  CALL T_CLEAN    ;
1130:   ;
1131:   ;
1132:  !********POSITIONER MOVE******** ;
1133:J P[811] 75% CNT25    ;
1134:   ;
1135:J P[812] 50% CNT80    ;
1136:   ;
1137:J P[813] 50% CNT30    ;
1138:   ;
1139:  !CELL ID: C ... ;
1140:   ;
1141:L P[814] 800mm/sec FINE
    :  Arc Start[1]    ;
1142:  WAIT    .15(sec) ;
1143:L P[815] WELD_SPEED FINE
    :  Arc End[1]    ;
1144:   ;
1145:J P[224] 50% CNT50    ;
1146:   ;
1147:L P[225] 800mm/sec FINE
    :  Arc Start[1]    ;
1148:  WAIT    .15(sec) ;
1149:L P[226] WELD_SPEED FINE
    :  Arc End[1]    ;
1150:   ;
1151:J P[227] 50% CNT50    ;
1152:   ;
1153:L P[228] 800mm/sec FINE
    :  Arc Start[1]    ;
1154:  WAIT    .15(sec) ;
1155:L P[229] WELD_SPEED FINE
    :  Arc End[1]    ;
1156:   ;
1157:J P[230] 50% CNT50    ;
1158:J P[816] 50% CNT60    ;
1159:   ;
1160:J P[817] 50% CNT80    ;
1161:   ;
1162:J P[818] 50% CNT60    ;
1163:   ;
1164:J P[819] 50% CNT60    ;
1165:   ;
1166:L P[820] 960mm/sec CNT25    ;
1167:   ;
1168:  !FR50X1650 ;
1169:  IF R[15]=1653,CALL TECH_HOLD ;
1170:   ;
1171:L P[821] 800mm/sec FINE
    :  Arc Start[6]    ;
1172:  Weave Sine[6] ;
1173:  Track TAST[6] ;
1174:L P[822] WELD_SPEED CNT100    ;
1175:C P[823]
    :  P[824] WELD_SPEED CNT100    ;
1176:L P[825] WELD_SPEED CNT100    ;
1177:C P[826]
    :  P[827] WELD_SPEED CNT100    ;
1178:L P[828] WELD_SPEED CNT100    ;
1179:L P[829] WELD_SPEED FINE
    :  Arc End[6]    ;
1180:  Weave End ;
1181:  Track End ;
1182:   ;
1183:L P[830] 1000mm/sec CNT25    ;
1184:   ;
1185:J P[831] 50% CNT25    ;
1186:   ;
1187:L P[832] 1000mm/sec CNT25    ;
1188:   ;
1189:   ;
1190:   ;
1191:  !FR50X1660 ;
1192:  !LENGTH: 40mm ;
1193:  ! ;
1194:  IF R[15]=1663,CALL TECH_HOLD ;
1195:   ;
1196:L P[833] 800mm/sec FINE
    :  Arc Start[6]    ;
1197:  Weave Sine[6] ;
1198:L P[834] WELD_SPEED FINE
    :  Arc End[6]    ;
1199:  Weave End ;
1200:   ;
1201:  CALL LENGTH_CHECK(1660) ;
1202:   ;
1203:L P[835] 1000mm/sec CNT25    ;
1204:   ;
1205:J P[842] 50% CNT10    ;
1206:   ;
1207:J P[843] 50% CNT10    ;
1208:   ;
1209:L P[844] 1000mm/sec CNT25    ;
1210:   ;
1211:  !FR50X1680 ;
1212:  IF R[15]=1683,CALL TECH_HOLD ;
1213:   ;
1214:L P[845] 800mm/sec FINE
    :  Arc Start[6]    ;
1215:  Weave Sine[6] ;
1216:  Track TAST[6] ;
1217:L P[846] WELD_SPEED FINE
    :  Arc End[6]    ;
1218:  Weave End ;
1219:  Track End ;
1220:   ;
1221:L P[847] 1000mm/sec CNT25    ;
1222:   ;
1223:  !********POSITIONER MOVE******** ;
1224:J P[848] 50% FINE    ;
1225:   ;
1226:  !FR50X1690 ;
1227:  IF R[15]=1693,CALL TECH_HOLD ;
1228:   ;
1229:L P[849] 800mm/sec FINE
    :  Arc Start[6]    ;
1230:  Weave Sine[6] ;
1231:  Track TAST[6] ;
1232:L P[850] WELD_SPEED CNT100    ;
1233:L P[851] WELD_SPEED CNT100    ;
1234:L P[852] WELD_SPEED CNT100    ;
1235:C P[853]
    :  P[854] WELD_SPEED CNT100    ;
1236:L P[855] WELD_SPEED CNT100    ;
1237:L P[856] WELD_SPEED CNT100    ;
1238:L P[857] WELD_SPEED CNT100    ;
1239:C P[858]
    :  P[859] WELD_SPEED CNT100    ;
1240:L P[860] WELD_SPEED CNT100    ;
1241:C P[861]
    :  P[862] WELD_SPEED CNT100    ;
1242:C P[863]
    :  P[864] WELD_SPEED CNT100    ;
1243:L P[865] WELD_SPEED FINE
    :  Arc End[6]    ;
1244:  Weave End ;
1245:  Track End ;
1246:   ;
1247:L P[866] 1000mm/sec CNT25    ;
1248:   ;
1249:L P[867] 1000mm/sec CNT25    ;
1250:   ;
1251:  !FR50X1700 ;
1252:  IF R[15]=1703,CALL TECH_HOLD ;
1253:   ;
1254:L P[868] 1000mm/sec FINE
    :  Arc Start[6]    ;
1255:  Weave Sine[6] ;
1256:  Track TAST[6] ;
1257:L P[869] WELD_SPEED CNT100    ;
1258:C P[870]
    :  P[871] WELD_SPEED CNT100    ;
1259:L P[872] WELD_SPEED CNT100    ;
1260:C P[873]
    :  P[874] WELD_SPEED CNT100    ;
1261:L P[875] WELD_SPEED CNT100    ;
1262:C P[876]
    :  P[877] WELD_SPEED CNT100    ;
1263:C P[878]
    :  P[879] WELD_SPEED FINE
    :  Arc End[6]    ;
1264:  Weave End ;
1265:  Track End ;
1266:   ;
1267:L P[880] 1000mm/sec CNT25    ;
1268:   ;
1269:L P[881] 1000mm/sec CNT25    ;
1270:   ;
1271:J P[882] 50% CNT25    ;
1272:   ;
1273:J P[883] 50% CNT25    ;
1274:   ;
1275:  !********POSITIONER MOVE******** ;
1276:J P[884] 75% FINE    ;
1277:   ;
1278:   ;
1279:  !FR50X1710 ;
1280:  IF R[15]=1713,CALL TECH_HOLD ;
1281:   ;
1282:L P[885] 800mm/sec FINE
    :  Arc Start[6]    ;
1283:  Weave Sine[6] ;
1284:  Track TAST[6] ;
1285:L P[236] WELD_SPEED CNT100    ;
1286:C P[886]
    :  P[887] WELD_SPEED CNT100    ;
1287:L P[888] WELD_SPEED CNT100    ;
1288:C P[889]
    :  P[890] WELD_SPEED CNT100    ;
1289:L P[891] WELD_SPEED FINE
    :  Arc End[6]    ;
1290:  Weave End ;
1291:  Track End ;
1292:   ;
1293:L P[892] 1000mm/sec CNT25    ;
1294:   ;
1295:J P[893] 50% CNT25    ;
1296:   ;
1297:  !FR50X1720 ;
1298:  IF R[15]=1723,CALL TECH_HOLD ;
1299:   ;
1300:L P[894] 800mm/sec FINE
    :  Arc Start[6]    ;
1301:  Weave Sine[6] ;
1302:  Track TAST[6] ;
1303:L P[895] WELD_SPEED CNT100    ;
1304:C P[896]
    :  P[897] WELD_SPEED CNT100    ;
1305:C P[898]
    :  P[899] WELD_SPEED CNT100    ;
1306:C P[900]
    :  P[901] WELD_SPEED CNT100    ;
1307:L P[902] WELD_SPEED FINE
    :  Arc End[6]    ;
1308:  Weave End ;
1309:  Track End ;
1310:   ;
1311:L P[903] 1000mm/sec CNT25    ;
1312:   ;
1313:L P[904] 500mm/sec CNT25    ;
1314:   ;
1315:L P[905] 500mm/sec CNT25    ;
1316:   ;
1317:   ;
1318:  !FR50X1730 ;
1319:  IF R[15]=1733,CALL TECH_HOLD ;
1320:   ;
1321:L P[906] 500mm/sec FINE
    :  Arc Start[6]    ;
1322:  Weave Sine[6] ;
1323:  Track TAST[6] ;
1324:L P[907] WELD_SPEED CNT100    ;
1325:L P[908] WELD_SPEED CNT100    ;
1326:L P[909] WELD_SPEED CNT100    ;
1327:L P[910] WELD_SPEED FINE
    :  Arc End[6]    ;
1328:  Weave End ;
1329:  Track End ;
1330:   ;
1331:L P[911] 500mm/sec CNT25    ;
1332:   ;
1333:L P[912] 1000mm/sec CNT25    ;
1334:   ;
1335:  !FR50X1740 ;
1336:  IF R[15]=1743,CALL TECH_HOLD ;
1337:   ;
1338:L P[913] 800mm/sec FINE
    :  Arc Start[6]    ;
1339:  Weave Sine[6] ;
1340:  Track TAST[6] ;
1341:L P[914] WELD_SPEED FINE
    :  Arc End[6]    ;
1342:  Weave End ;
1343:  Track End ;
1344:   ;
1345:L P[915] 960mm/sec CNT40    ;
1346:   ;
1347:J P[916] 50% CNT35    ;
1348:   ;
1349:  !FR50X1750 ;
1350:  IF R[15]=1753,CALL TECH_HOLD ;
1351:   ;
1352:L P[917] 800mm/sec FINE
    :  Arc Start[6]    ;
1353:  Weave Sine[6] ;
1354:L P[918] WELD_SPEED FINE
    :  Arc End[6]    ;
1355:  Weave End ;
1356:   ;
1357:L P[919] 1000mm/sec CNT50    ;
1358:   ;
1359:J P[223] 50% CNT25    ;
1360:   ;
1361:J P[920] 50% CNT25    ;
1362:   ;
1363:  !FR50X1760 ;
1364:  IF R[15]=1763,CALL TECH_HOLD ;
1365:   ;
1366:L P[921] 800mm/sec FINE
    :  Arc Start[6]    ;
1367:  Weave Sine[6] ;
1368:  Track TAST[6] ;
1369:L P[922] WELD_SPEED FINE
    :  Arc End[6]    ;
1370:  Weave End ;
1371:  Track End ;
1372:   ;
1373:L P[923] 500mm/sec CNT25    ;
1374:   ;
1375:J P[924] 50% CNT25    ;
1376:   ;
1377:J P[925] 50% CNT25    ;
1378:   ;
1379:   ;
1380:  !FR50X1770 ;
1381:  IF R[15]=1773,CALL TECH_HOLD ;
1382:   ;
1383:   ;
1384:L P[926] 1000mm/sec FINE
    :  Arc Start[6]    ;
1385:  Weave Sine[6] ;
1386:  Track TAST[6] ;
1387:L P[927] WELD_SPEED FINE
    :  Arc End[6]    ;
1388:  Weave End ;
1389:  Track End ;
1390:   ;
1391:L P[928] 1000mm/sec CNT25    ;
1392:   ;
1393:L P[929] 1000mm/sec CNT25    ;
1394:   ;
1395:J P[930] 50% CNT25    ;
1396:   ;
1397:   ;
1398:  !FR50X1780 ;
1399:  IF R[15]=1783,CALL TECH_HOLD ;
1400:   ;
1401:L P[931] 1000mm/sec FINE
    :  Arc Start[6]    ;
1402:  Weave Sine[6] ;
1403:  Track TAST[6] ;
1404:L P[932] WELD_SPEED FINE
    :  Arc End[6]    ;
1405:  Weave End ;
1406:  Track End ;
1407:   ;
1408:L P[933] 1000mm/sec CNT25    ;
1409:   ;
1410:J P[934] 50% CNT45    ;
1411:   ;
1412:J P[935] 50% CNT40    ;
1413:   ;
1414:  !********POSITIONER MOVE******** ;
1415:J P[936] 80% CNT25    ;
1416:   ;
1417:J P[937] 50% CNT40    ;
1418:   ;
1419:J P[938] 25% CNT15    ;
1420:   ;
1421:L P[231] 450mm/sec CNT25    ;
1422:   ;
1423:  CALL ARC_DISABLE_RH_LS(0) ;
1424:   ;
1425:  !FR50X1790 ;
1426:  IF R[15]=1793,CALL TECH_HOLD ;
1427:   ;
1428:L P[939] 200mm/sec FINE
    :  Arc Start[8]    ;
1429:  Weave Sine[8] ;
1430:L P[940] WELD_SPEED CNT100    ;
1431:C P[941]
    :  P[942] WELD_SPEED CNT100    ;
1432:L P[943] WELD_SPEED FINE
    :  Arc End[8]    ;
1433:  Weave End ;
1434:   ;
1435:L P[944] 200mm/sec CNT15    ;
1436:   ;
1437:J P[945] 50% CNT25    ;
1438:   ;
1439:  !FR50X1800 ;
1440:  IF R[15]=1803,CALL TECH_HOLD ;
1441:   ;
1442:L P[946] 300mm/sec FINE
    :  Arc Start[8]    ;
1443:  Weave Sine[8] ;
1444:L P[947] WELD_SPEED FINE
    :  Arc End[8]    ;
1445:  Weave End ;
1446:   ;
1447:  CALL ARC_DISABLE_RH_LS(1) ;
1448:   ;
1449:L P[948] 300mm/sec CNT25    ;
1450:   ;
1451:J P[949] 50% CNT25    ;
1452:   ;
1453:  !HOME ;
1454:J P[950] 100% CNT25    ;
1455:   ;
1456:  !TORCH CLEAN ;
1457:  CALL HOME    ;
1458:  CALL T_CLEAN    ;
1459:   ;
1460:  !********POSITIONER MOVE******** ;
1461:J P[951] 75% FINE    ;
1462:   ;
1463:J P[952] 50% CNT25    ;
1464:   ;
1465:L P[953] 1000mm/sec CNT25    ;
1466:   ;
1467:  !FR50X1810 ;
1468:  IF R[15]=1813,CALL TECH_HOLD ;
1469:   ;
1470:L P[954] 800mm/sec FINE
    :  Arc Start[6]    ;
1471:  Weave Sine[6] ;
1472:  Track TAST[6] ;
1473:L P[955] WELD_SPEED FINE
    :  Arc End[6]    ;
1474:  Weave End ;
1475:  Track End ;
1476:   ;
1477:L P[956] 300mm/sec CNT25    ;
1478:   ;
1479:L P[957] 1000mm/sec CNT25    ;
1480:   ;
1481:J P[958] 50% CNT25    ;
1482:   ;
1483:J P[959] 50% CNT25    ;
1484:   ;
1485:L P[960] 1000mm/sec CNT25    ;
1486:   ;
1487:  !FR50X1820 ;
1488:  IF R[15]=1823,CALL TECH_HOLD ;
1489:   ;
1490:L P[961] 1000mm/sec FINE
    :  Arc Start[6]    ;
1491:  Weave Sine[6] ;
1492:  Track TAST[6] ;
1493:C P[962]
    :  P[963] WELD_SPEED CNT100    ;
1494:L P[964] WELD_SPEED FINE
    :  Arc End[6]    ;
1495:  Weave End ;
1496:  Track End ;
1497:   ;
1498:L P[965] 300mm/sec CNT25    ;
1499:   ;
1500:L P[966] 1000mm/sec CNT25    ;
1501:   ;
1502:  !HOME ;
1503:J P[967] 100% CNT25    ;
1504:   ;
1505:  !********POSITIONER MOVE******** ;
1506:J P[968] 75% FINE    ;
1507:   ;
1508:L P[969] 1000mm/sec CNT25    ;
1509:   ;
1510:  !FR50X1830 ;
1511:  IF R[15]=1833,CALL TECH_HOLD ;
1512:   ;
1513:L P[970] 1000mm/sec FINE
    :  Arc Start[6]    ;
1514:  Weave Sine[6] ;
1515:  Track TAST[6] ;
1516:C P[971]
    :  P[972] WELD_SPEED CNT100    ;
1517:L P[973] WELD_SPEED FINE
    :  Arc End[6]    ;
1518:  Weave End ;
1519:  Track End ;
1520:   ;
1521:L P[974] 300mm/sec CNT25    ;
1522:   ;
1523:L P[975] 1000mm/sec CNT25    ;
1524:   ;
1525:  !HOME ;
1526:J P[976] 100% FINE    ;
1527:   ;
1528:  !********POSITIONER MOVE******** ;
1529:J P[977] 75% CNT25    ;
1530:   ;
1531:J P[978] 50% CNT25    ;
1532:   ;
1533:L P[979] 1000mm/sec CNT25    ;
1534:   ;
1535:  //UALM[20] ;
1536:  !DOUBLE CHECK ;
1537:   ;
1538:   ;
1539:  !FR50X1840 ;
1540:  !LENGTH: 40mm ;
1541:   ;
1542:  IF R[15]=1843,CALL TECH_HOLD ;
1543:   ;
1544:L P[980] 800mm/sec FINE
    :  Arc Start[6]    ;
1545:  Weave Sine[6] ;
1546:L P[981] WELD_SPEED FINE
    :  Arc End[6]    ;
1547:  Weave End ;
1548:   ;
1549:  CALL LENGTH_CHECK(1840) ;
1550:   ;
1551:L P[982] 1000mm/sec CNT25    ;
1552:   ;
1553:L P[983] 1000mm/sec CNT25    ;
1554:   ;
1555:J P[984] 50% CNT25    ;
1556:   ;
1557:L P[985] 1000mm/sec CNT25    ;
1558:   ;
1559:  !FR50X1850 ;
1560:  IF R[15]=1853,CALL TECH_HOLD ;
1561:   ;
1562:L P[986] 800mm/sec FINE
    :  Arc Start[6]    ;
1563:  Weave Sine[6] ;
1564:L P[987] WELD_SPEED CNT100    ;
1565:C P[988]
    :  P[989] WELD_SPEED FINE
    :  Arc End[6]    ;
1566:  Weave End ;
1567:   ;
1568:L P[990] 500mm/sec CNT25    ;
1569:   ;
1570:L P[991] 1000mm/sec CNT25    ;
1571:   ;
1572:J P[992] 50% CNT25    ;
1573:   ;
1574:L P[993] 1000mm/sec CNT25    ;
1575:   ;
1576:L P[994] 500mm/sec CNT25    ;
1577:   ;
1578:  !FR50X1860 ;
1579:  IF R[15]=1863,CALL TECH_HOLD ;
1580:   ;
1581:L P[995] 800mm/sec FINE
    :  Arc Start[6]    ;
1582:  Weave Sine[6] ;
1583:L P[996] WELD_SPEED CNT100    ;
1584:C P[997]
    :  P[998] WELD_SPEED FINE
    :  Arc End[6]    ;
1585:  Weave End ;
1586:   ;
1587:L P[999] 300mm/sec CNT5    ;
1588:   ;
1589:L P[1000] 500mm/sec CNT5    ;
1590:   ;
1591:L P[1001] 1000mm/sec CNT25    ;
1592:   ;
1593:J P[1002] 50% CNT25    ;
1594:   ;
1595:L P[1003] 1000mm/sec CNT25    ;
1596:   ;
1597:  !FR50X1870 ;
1598:  IF R[15]=1873,CALL TECH_HOLD ;
1599:   ;
1600:L P[1004] 800mm/sec FINE
    :  Arc Start[6]    ;
1601:  Weave Sine[6] ;
1602:  Track TAST[6] ;
1603:C P[1005]
    :  P[1006] WELD_SPEED CNT100    ;
1604:L P[1007] WELD_SPEED CNT100    ;
1605:C P[1008]
    :  P[1009] WELD_SPEED CNT100    ;
1606:L P[1010] WELD_SPEED CNT100    ;
1607:C P[1011]
    :  P[1012] WELD_SPEED CNT100    ;
1608:L P[1013] WELD_SPEED FINE
    :  Arc End[6]    ;
1609:  Weave End ;
1610:  Track End ;
1611:   ;
1612:L P[1014] 1000mm/sec CNT50    ;
1613:   ;
1614:J P[1015] 50% CNT10    ;
1615:   ;
1616:L P[1016] 1000mm/sec CNT25    ;
1617:   ;
1618:  !FR50X1880 ;
1619:  IF R[15]=1883,CALL TECH_HOLD ;
1620:   ;
1621:L P[1017] 800mm/sec FINE
    :  Arc Start[6]    ;
1622:  Weave Sine[6] ;
1623:  Track TAST[6] ;
1624:L P[1018] WELD_SPEED FINE
    :  Arc End[6]    ;
1625:  Weave End ;
1626:  Track End ;
1627:   ;
1628:L P[1019] 1000mm/sec CNT25    ;
1629:   ;
1630:  !********POSITIONER MOVE******** ;
1631:J P[1020] 75% FINE    ;
1632:   ;
1633:  !FR50X1890 ;
1634:  IF R[15]=1893,CALL TECH_HOLD ;
1635:   ;
1636:L P[1021] 800mm/sec FINE
    :  Arc Start[6]    ;
1637:  Weave Sine[6] ;
1638:  Track TAST[6] ;
1639:L P[1022] WELD_SPEED CNT100    ;
1640:C P[1023]
    :  P[1024] WELD_SPEED CNT100    ;
1641:L P[1025] WELD_SPEED CNT100    ;
1642:C P[1026]
    :  P[1027] WELD_SPEED CNT100    ;
1643:L P[1028] WELD_SPEED CNT100    ;
1644:C P[1029]
    :  P[1030] WELD_SPEED CNT100    ;
1645:L P[1031] WELD_SPEED FINE
    :  Arc End[6]    ;
1646:  Weave End ;
1647:  Track End ;
1648:   ;
1649:L P[1032] 1000mm/sec CNT25    ;
1650:   ;
1651:L P[1033] 1000mm/sec CNT25    ;
1652:   ;
1653:  !FR50X1900 ;
1654:  IF R[15]=1903,CALL TECH_HOLD ;
1655:   ;
1656:L P[1034] 800mm/sec FINE
    :  Arc Start[6]    ;
1657:  Weave Sine[6] ;
1658:  Track TAST[6] ;
1659:L P[1035] WELD_SPEED CNT100    ;
1660:C P[1036]
    :  P[1037] WELD_SPEED CNT100    ;
1661:L P[1038] WELD_SPEED CNT100    ;
1662:C P[1039]
    :  P[1040] WELD_SPEED CNT100    ;
1663:L P[1041] WELD_SPEED CNT100    ;
1664:C P[1042]
    :  P[1043] WELD_SPEED CNT100    ;
1665:C P[1044]
    :  P[1045] WELD_SPEED FINE
    :  Arc End[6]    ;
1666:  Weave End ;
1667:  Track End ;
1668:   ;
1669:L P[1046] 1000mm/sec CNT25    ;
1670:   ;
1671:L P[1047] 1000mm/sec CNT25    ;
1672:   ;
1673:L P[1048] 1000mm/sec CNT25    ;
1674:   ;
1675:L P[1049] 1000mm/sec CNT25    ;
1676:   ;
1677:  !HOME ;
1678:J P[1050] 100% FINE    ;
1679:   ;
1680:  !********POSITIONER MOVE******** ;
1681:J P[1051] 50% CNT25    ;
1682:   ;
1683:  !FR50X1910 ;
1684:  IF R[15]=1913,CALL TECH_HOLD ;
1685:   ;
1686:L P[1052] 780mm/sec FINE
    :  Arc Start[6]    ;
1687:  Weave Sine[6] ;
1688:  Track TAST[6] ;
1689:L P[1053] WELD_SPEED CNT100    ;
1690:C P[1054]
    :  P[1055] WELD_SPEED CNT100    ;
1691:L P[1056] WELD_SPEED CNT100    ;
1692:C P[1057]
    :  P[1058] WELD_SPEED FINE
    :  Arc End[6]    ;
1693:  Weave End ;
1694:  Track End ;
1695:   ;
1696:L P[1059] 1000mm/sec CNT25    ;
1697:   ;
1698:J P[1060] 50% CNT25    ;
1699:   ;
1700:  !FR50X1920 ;
1701:  IF R[15]=1923,CALL TECH_HOLD ;
1702:   ;
1703:L P[1061] 800mm/sec FINE
    :  Arc Start[6]    ;
1704:  Weave Sine[6] ;
1705:  Track TAST[6] ;
1706:L P[1062] WELD_SPEED CNT100    ;
1707:C P[1063]
    :  P[1064] WELD_SPEED CNT100    ;
1708:C P[1065]
    :  P[1066] WELD_SPEED CNT100    ;
1709:C P[1067]
    :  P[1068] WELD_SPEED CNT100    ;
1710:L P[1069] WELD_SPEED FINE
    :  Arc End[6]    ;
1711:  Weave End ;
1712:  Track End ;
1713:   ;
1714:L P[1070] 1000mm/sec CNT25    ;
1715:   ;
1716:L P[1071] 1000mm/sec CNT25    ;
1717:   ;
1718:  !FR50X1930 ;
1719:  IF R[15]=1933,CALL TECH_HOLD ;
1720:   ;
1721:L P[1072] 800mm/sec FINE
    :  Arc Start[6]    ;
1722:  Weave Sine[6] ;
1723:  Track TAST[6] ;
1724:L P[1073] WELD_SPEED FINE
    :  Arc End[6]    ;
1725:  Weave End ;
1726:  Track End ;
1727:   ;
1728:L P[1074] 1000mm/sec CNT25    ;
1729:   ;
1730:L P[1075] 1000mm/sec CNT50    ;
1731:   ;
1732:  !FR50X1940 ;
1733:  IF R[15]=1943,CALL TECH_HOLD ;
1734:   ;
1735:L P[1076] 800mm/sec FINE
    :  Arc Start[6]    ;
1736:  Weave Sine[6] ;
1737:L P[1077] WELD_SPEED FINE
    :  Arc End[6]    ;
1738:  Weave End ;
1739:   ;
1740:L P[1078] 1000mm/sec CNT50    ;
1741:   ;
1742:J P[1079] 50% CNT25    ;
1743:   ;
1744:  !FR50X1950 ;
1745:  IF R[15]=1953,CALL TECH_HOLD ;
1746:   ;
1747:L P[1080] 800mm/sec FINE
    :  Arc Start[6]    ;
1748:  Weave Sine[6] ;
1749:  Track TAST[6] ;
1750:L P[1081] WELD_SPEED FINE
    :  Arc End[6]    ;
1751:  Weave End ;
1752:  Track End ;
1753:   ;
1754:L P[1082] 1000mm/sec CNT25    ;
1755:   ;
1756:J P[1083] 50% CNT25    ;
1757:   ;
1758:J P[1084] 50% CNT25    ;
1759:   ;
1760:  !FR50X1960 ;
1761:  IF R[15]=1963,CALL TECH_HOLD ;
1762:   ;
1763:L P[1085] 800mm/sec FINE
    :  Arc Start[6]    ;
1764:  Weave Sine[6] ;
1765:L P[1086] WELD_SPEED FINE
    :  Arc End[6]    ;
1766:  Weave End ;
1767:   ;
1768:L P[1087] 1000mm/sec CNT100    ;
1769:   ;
1770:J P[1088] 50% CNT30    ;
1771:   ;
1772:  !FR50X1970 ;
1773:  IF R[15]=1973,CALL TECH_HOLD ;
1774:   ;
1775:L P[1089] 780mm/sec FINE
    :  Arc Start[6]    ;
1776:  Weave Sine[6] ;
1777:L P[1090] WELD_SPEED FINE
    :  Arc End[6]    ;
1778:  Weave End ;
1779:   ;
1780:L P[1091] 1000mm/sec CNT75    ;
1781:   ;
1782:J P[1092] 50% CNT40    ;
1783:   ;
1784:  !********POSITIONER MOVE******** ;
1785:J P[1093] 75% CNT25    ;
1786:   ;
1787:J P[1094] 50% CNT25    ;
1788:   ;
1789:J P[1095] 50% CNT30    ;
1790:   ;
1791:L P[1096] 1000mm/sec CNT70    ;
1792:   ;
1793:L P[232] 500mm/sec CNT50    ;
1794:   ;
1795:  CALL ARC_LH_DISABLE_LS(0) ;
1796:   ;
1797:  !FR50X1980 ;
1798:  IF R[15]=1983,CALL TECH_HOLD ;
1799:   ;
1800:L P[1097] 200mm/sec FINE
    :  Arc Start[8]    ;
1801:  Weave Sine[8] ;
1802:L P[1098] WELD_SPEED CNT100    ;
1803:C P[1099]
    :  P[1100] WELD_SPEED CNT100    ;
1804:L P[1101] WELD_SPEED FINE
    :  Arc End[8]    ;
1805:  Weave End ;
1806:   ;
1807:J P[1102] 50% CNT40    ;
1808:   ;
1809:J P[1103] 50% CNT70    ;
1810:   ;
1811:J P[1104] 50% CNT35    ;
1812:   ;
1813:  !FR50X1990 ;
1814:  IF R[15]=1993,CALL TECH_HOLD ;
1815:   ;
1816:L P[1105] 800mm/sec FINE
    :  Arc Start[8]    ;
1817:  Weave Sine[8] ;
1818:L P[1106] WELD_SPEED FINE
    :  Arc End[8]    ;
1819:  Weave End ;
1820:   ;
1821:  CALL ARC_LH_DISABLE_LS(1) ;
1822:   ;
1823:J P[1107] 25% CNT40    ;
1824:   ;
1825:J P[1108] 50% CNT25    ;
1826:   ;
1827:J P[1109] 50% CNT50    ;
1828:   ;
1829:  !HOME ;
1830:J P[1110] 100% CNT25    ;
1831:   ;
1832:  !********POSITIONER MOVE******** ;
1833:J P[1111] 75% FINE    ;
1834:   ;
1835:J P[1112] 50% CNT25    ;
1836:   ;
1837:L P[1113] 1000mm/sec CNT25    ;
1838:   ;
1839:L P[1114] 500mm/sec CNT25    ;
1840:   ;
1841:  !FR50X2000 ;
1842:  IF R[15]=2003,CALL TECH_HOLD ;
1843:   ;
1844:L P[1115] 800mm/sec FINE
    :  Arc Start[6]    ;
1845:  Weave Sine[6] ;
1846:L P[1116] WELD_SPEED FINE
    :  Arc End[6]    ;
1847:  Weave End ;
1848:   ;
1849:L P[1117] 500mm/sec CNT25    ;
1850:   ;
1851:L P[1118] 1000mm/sec CNT25    ;
1852:   ;
1853:J P[1119] 50% CNT25    ;
1854:   ;
1855:   ;
1856:  CALL HOME    ;
1857:  CALL LOAD_POS    ;
1858:   ;
/POS
P[1]{
   GP1:
	UF : 1, UT : 1,		CONFIG : 'N U T, 0, 0, 0',
	X =  1214.464  mm,	Y =  1589.090  mm,	Z =   593.946  mm,
	W =      .000 deg,	P =    44.876 deg,	R =   135.007 deg
   GP2:
	UF : 0, UT : 1,
	J1=     0.000 deg,	J2=    45.000 deg
};
P[2]{
   GP1:
	UF : 1, UT : 1,		CONFIG : 'N U T, 0, 0, 0',
	X =  1343.971  mm,	Y =  1452.300  mm,	Z =   232.946  mm,
	W =      .000 deg,	P =    44.876 deg,	R =   135.007 deg
   GP2:
	UF : 0, UT : 1,
	J1=     0.000 deg,	J2=    45.000 deg
};
P[3]{
   GP1:
	UF : 1, UT : 1,		CONFIG : 'N U T, 0, 0, 0',
	X =  1390.272  mm,	Y =  1354.500  mm,	Z =    79.223  mm,
	W =      .004 deg,	P =    44.873 deg,	R =   131.158 deg
   GP2:
	UF : 0, UT : 1,
	J1=     0.000 deg,	J2=    45.000 deg
};
P[4]{
   GP1:
	UF : 1, UT : 1,		CONFIG : 'N U T, 0, 0, 0',
	X =  1442.813  mm,	Y =  1410.035  mm,	Z =    81.944  mm,
	W =     -.001 deg,	P =    44.845 deg,	R =   152.019 deg
   GP2:
	UF : 0, UT : 1,
	J1=     0.000 deg,	J2=    45.000 deg
};
P[5]{
   GP1:
	UF : 1, UT : 1,		CONFIG : 'N U T, 0, 0, 0',
	X =  1406.269  mm,	Y =  1426.258  mm,	Z =   124.762  mm,
	W =     -.002 deg,	P =    44.845 deg,	R =   152.019 deg
   GP2:
	UF : 0, UT : 1,
	J1=     0.000 deg,	J2=    45.000 deg
};
P[6]{
   GP1:
	UF : 1, UT : 1,		CONFIG : 'N U T, 0, 0, 0',
	X =  1327.201  mm,	Y =  1350.025  mm,	Z =   146.947  mm,
	W =     -.000 deg,	P =    44.876 deg,	R =   131.152 deg
   GP2:
	UF : 0, UT : 1,
	J1=     0.000 deg,	J2=    45.000 deg
};
P[7]{
   GP1:
	UF : 1, UT : 1,		CONFIG : 'N U T, 0, 0, 0',
	X =  1360.318  mm,	Y =  1328.105  mm,	Z =    81.017  mm,
	W =      .000 deg,	P =    44.876 deg,	R =   131.152 deg
   GP2:
	UF : 0, UT : 1,
	J1=     0.000 deg,	J2=    45.000 deg
};
P[8]{
   GP1:
	UF : 1, UT : 1,		CONFIG : 'N U T, 0, 0, 0',
	X =   968.269  mm,	Y =   941.123  mm,	Z =    79.601  mm,
	W =      .000 deg,	P =    44.876 deg,	R =   127.977 deg
   GP2:
	UF : 0, UT : 1,
	J1=     0.000 deg,	J2=    45.000 deg
};
P[9]{
   GP1:
	UF : 1, UT : 1,		CONFIG : 'N U T, 0, 0, 0',
	X =   922.593  mm,	Y =   918.484  mm,	Z =   118.901  mm,
	W =     -.000 deg,	P =    44.876 deg,	R =   129.337 deg
   GP2:
	UF : 0, UT : 1,
	J1=     0.000 deg,	J2=    45.000 deg
};
P[10]{
   GP1:
	UF : 1, UT : 1,		CONFIG : 'N U T, 0, 0, 0',
	X =   932.883  mm,	Y =   905.922  mm,	Z =    80.529  mm,
	W =      .005 deg,	P =    44.838 deg,	R =   129.334 deg
   GP2:
	UF : 0, UT : 1,
	J1=     0.000 deg,	J2=    45.000 deg
};
P[11]{
   GP1:
	UF : 1, UT : 1,		CONFIG : 'N U T, 0, 0, 0',
	X =   885.701  mm,	Y =   855.031  mm,	Z =    77.818  mm,
	W =      .000 deg,	P =    44.876 deg,	R =   129.337 deg
   GP2:
	UF : 0, UT : 1,
	J1=     0.000 deg,	J2=    45.000 deg
};
P[12]{
   GP1:
	UF : 1, UT : 1,		CONFIG : 'N U T, 0, 0, 0',
	X =   879.676  mm,	Y =   853.017  mm,	Z =    79.876  mm,
	W =      .003 deg,	P =    44.796 deg,	R =   114.722 deg
   GP2:
	UF : 0, UT : 1,
	J1=     0.000 deg,	J2=    45.000 deg
};
P[13]{
   GP1:
	UF : 1, UT : 1,		CONFIG : 'N U T, 0, 0, 0',
	X =   863.490  mm,	Y =   904.621  mm,	Z =   146.286  mm,
	W =      .000 deg,	P =    44.876 deg,	R =   112.101 deg
   GP2:
	UF : 0, UT : 1,
	J1=     0.000 deg,	J2=    45.000 deg
};
P[14]{
   GP1:
	UF : 1, UT : 1,		CONFIG : 'N U T, 0, 0, 0',
	X =   831.040  mm,	Y =  1277.928  mm,	Z =   275.925  mm,
	W =      .000 deg,	P =    44.876 deg,	R =   112.101 deg
   GP2:
	UF : 0, UT : 1,
	J1=     0.000 deg,	J2=    45.000 deg
};
P[15]{
   GP1:
	UF : 1, UT : 1,		CONFIG : 'N U B, 0, 0, 0',
	X =   353.784  mm,	Y =     3.997  mm,	Z =  2425.735  mm,
	W =     -.021 deg,	P =   -39.773 deg,	R =      .020 deg
   GP2:
	UF : 1, UT : 1,
	J1=     0.000 deg,	J2=    45.000 deg
};
P[16]{
   GP1:
	UF : 1, UT : 1,
	J1=    -2.565 deg,	J2=   -47.918 deg,	J3=    37.877 deg,
	J4=   -63.535 deg,	J5=   -19.106 deg,	J6=    56.044 deg
   GP2:
	UF : 0, UT : 1,
	J1=     0.000 deg,	J2=   180.000 deg
};
P[17]{
   GP1:
	UF : 1, UT : 1,		CONFIG : 'N U T, 0, 0, 0',
	X =  2036.678  mm,	Y =   133.789  mm,	Z =  1445.358  mm,
	W =   -25.929 deg,	P =   -45.424 deg,	R =    36.423 deg
   GP2:
	UF : 0, UT : 1,
	J1=     0.000 deg,	J2=   180.000 deg
};
P[18]{
   GP1:
	UF : 1, UT : 1,		CONFIG : 'N U T, 0, 0, 0',
	X =  2233.304  mm,	Y =   372.944  mm,	Z =  1162.580  mm,
	W =   -27.414 deg,	P =   -38.078 deg,	R =    43.574 deg
   GP2:
	UF : 0, UT : 1,
	J1=     0.000 deg,	J2=   180.000 deg
};
P[19]{
   GP1:
	UF : 1, UT : 1,		CONFIG : 'N U T, 0, 0, 0',
	X =  2281.974  mm,	Y =   431.829  mm,	Z =  1116.684  mm,
	W =   -41.778 deg,	P =   -28.391 deg,	R =    61.958 deg
   GP2:
	UF : 0, UT : 1,
	J1=      .000 deg,	J2=   180.000 deg
};
P[20]{
   GP1:
	UF : 1, UT : 1,		CONFIG : 'N U T, 0, 0, 0',
	X =  2287.244  mm,	Y =    94.810  mm,	Z =  1116.986  mm,
	W =   -31.951 deg,	P =   -39.356 deg,	R =    44.493 deg
   GP2:
	UF : 0, UT : 1,
	J1=      .000 deg,	J2=   180.000 deg
};
P[21]{
   GP1:
	UF : 1, UT : 1,		CONFIG : 'N U T, 0, 0, 0',
	X =  2124.976  mm,	Y =    85.873  mm,	Z =  1194.632  mm,
	W =   -28.024 deg,	P =   -38.698 deg,	R =    43.953 deg
   GP2:
	UF : 0, UT : 1,
	J1=     0.000 deg,	J2=   180.000 deg
};
P[22]{
   GP1:
	UF : 1, UT : 1,		CONFIG : 'N U T, 0, 0, 0',
	X =  2124.976  mm,	Y =  -285.127  mm,	Z =  1194.632  mm,
	W =    36.159 deg,	P =   -31.426 deg,	R =   -50.949 deg
   GP2:
	UF : 0, UT : 1,
	J1=     0.000 deg,	J2=   180.000 deg
};
P[23]{
   GP1:
	UF : 1, UT : 1,		CONFIG : 'N U T, 0, 0, 0',
	X =  2228.976  mm,	Y =  -404.127  mm,	Z =  1194.631  mm,
	W =    36.159 deg,	P =   -31.426 deg,	R =   -50.949 deg
   GP2:
	UF : 0, UT : 1,
	J1=     0.000 deg,	J2=   180.000 deg
};
P[24]{
   GP1:
	UF : 1, UT : 1,		CONFIG : 'N U T, 0, 0, 0',
	X =  2286.216  mm,	Y =  -430.685  mm,	Z =  1116.208  mm,
	W =    43.325 deg,	P =   -25.600 deg,	R =   -65.383 deg
   GP2:
	UF : 0, UT : 1,
	J1=      .000 deg,	J2=   180.000 deg
};
P[25]{
   GP1:
	UF : 1, UT : 1,		CONFIG : 'N U T, 0, 0, 0',
	X =  2285.704  mm,	Y =   -96.057  mm,	Z =  1118.736  mm,
	W =    36.109 deg,	P =   -35.685 deg,	R =   -49.851 deg
   GP2:
	UF : 0, UT : 1,
	J1=      .000 deg,	J2=   180.000 deg
};
P[26]{
   GP1:
	UF : 1, UT : 1,		CONFIG : 'N U T, 0, 0, 0',
	X =  2200.047  mm,	Y =  -119.764  mm,	Z =  1205.936  mm,
	W =    36.159 deg,	P =   -31.426 deg,	R =   -50.949 deg
   GP2:
	UF : 0, UT : 1,
	J1=     0.000 deg,	J2=   180.000 deg
};
P[27]{
   GP1:
	UF : 1, UT : 1,		CONFIG : 'N U T, 0, 0, 0',
	X =  2148.046  mm,	Y =   213.236  mm,	Z =  1205.936  mm,
	W =    43.692 deg,	P =    17.672 deg,	R =   -14.083 deg
   GP2:
	UF : 0, UT : 1,
	J1=     0.000 deg,	J2=   180.000 deg
};
P[28]{
   GP1:
	UF : 1, UT : 1,		CONFIG : 'N U T, 0, 0, 0',
	X =  2215.047  mm,	Y =   399.236  mm,	Z =  1133.936  mm,
	W =    46.448 deg,	P =     -.794 deg,	R =    -1.597 deg
   GP2:
	UF : 0, UT : 1,
	J1=     0.000 deg,	J2=   180.000 deg
};
P[29]{
   GP1:
	UF : 1, UT : 1,		CONFIG : 'N U T, 0, 0, 0',
	X =  2267.390  mm,	Y =   445.167  mm,	Z =  1114.198  mm,
	W =    45.219 deg,	P =     6.865 deg,	R =   -26.427 deg
   GP2:
	UF : 0, UT : 1,
	J1=      .000 deg,	J2=   180.000 deg
};
P[30]{
   GP1:
	UF : 1, UT : 1,		CONFIG : 'N U T, 0, 0, 0',
	X =  2216.474  mm,	Y =   448.477  mm,	Z =  1105.205  mm,
	W =    45.349 deg,	P =    -4.892 deg,	R =    -3.107 deg
   GP2:
	UF : 0, UT : 1,
	J1=     0.000 deg,	J2=   180.000 deg
};
P[31]{
   GP1:
	UF : 1, UT : 1,		CONFIG : 'N U T, 0, 0, 0',
	X =  1802.457  mm,	Y =   450.063  mm,	Z =  1048.114  mm,
	W =    45.349 deg,	P =    -4.892 deg,	R =    -3.106 deg
   GP2:
	UF : 0, UT : 1,
	J1=     0.000 deg,	J2=   180.000 deg
};
P[32]{
   GP1:
	UF : 1, UT : 1,		CONFIG : 'N U T, 0, 0, 0',
	X =  1805.495  mm,	Y =   305.433  mm,	Z =  1168.972  mm,
	W =    45.922 deg,	P =    -2.604 deg,	R =     -.767 deg
   GP2:
	UF : 0, UT : 1,
	J1=     0.000 deg,	J2=   180.000 deg
};
P[33]{
   GP1:
	UF : 1, UT : 1,		CONFIG : 'N U T, 0, 0, 0',
	X =  1924.292  mm,	Y =   -66.744  mm,	Z =  1269.461  mm,
	W =   -12.797 deg,	P =    45.048 deg,	R =    98.836 deg
   GP2:
	UF : 0, UT : 1,
	J1=     0.000 deg,	J2=   180.000 deg
};
P[34]{
   GP1:
	UF : 1, UT : 1,		CONFIG : 'N U T, 0, 0, 0',
	X =  2240.823  mm,	Y =  -392.629  mm,	Z =  1154.975  mm,
	W =   -42.742 deg,	P =    20.262 deg,	R =    31.070 deg
   GP2:
	UF : 0, UT : 1,
	J1=     0.000 deg,	J2=   180.000 deg
};
P[35]{
   GP1:
	UF : 1, UT : 1,		CONFIG : 'N U T, 0, 0, 0',
	X =  2264.216  mm,	Y =  -448.220  mm,	Z =  1113.311  mm,
	W =   -44.574 deg,	P =    10.493 deg,	R =    27.731 deg
   GP2:
	UF : 0, UT : 1,
	J1=      .000 deg,	J2=   180.000 deg
};
P[36]{
   GP1:
	UF : 1, UT : 1,		CONFIG : 'N U T, 0, 0, 0',
	X =  2224.221  mm,	Y =  -446.957  mm,	Z =  1106.872  mm,
	W =   -43.356 deg,	P =    15.621 deg,	R =    23.835 deg
   GP2:
	UF : 0, UT : 1,
	J1=     0.000 deg,	J2=   180.000 deg
};
P[37]{
   GP1:
	UF : 1, UT : 1,		CONFIG : 'N U T, 0, 0, 0',
	X =  1800.140  mm,	Y =  -448.282  mm,	Z =  1046.276  mm,
	W =   -38.710 deg,	P =    26.186 deg,	R =    36.762 deg
   GP2:
	UF : 0, UT : 1,
	J1=     0.000 deg,	J2=   180.000 deg
};
P[38]{
   GP1:
	UF : 1, UT : 1,		CONFIG : 'N U T, 0, 0, 0',
	X =  1821.930  mm,	Y =  -324.610  mm,	Z =  1168.225  mm,
	W =   -42.742 deg,	P =    20.262 deg,	R =    19.276 deg
   GP2:
	UF : 0, UT : 1,
	J1=     0.000 deg,	J2=   180.000 deg
};
P[39]{
   GP1:
	UF : 1, UT : 1,		CONFIG : 'N U T, 0, 0, 0',
	X =  1912.048  mm,	Y =   149.237  mm,	Z =   872.936  mm,
	W =    45.096 deg,	P =    12.591 deg,	R =   -12.476 deg
   GP2:
	UF : 0, UT : 1,
	J1=     0.000 deg,	J2=   180.000 deg
};
P[40]{
   GP1:
	UF : 1, UT : 1,		CONFIG : 'N U T, 0, 0, 0',
	X =  2084.488  mm,	Y =   344.809  mm,	Z =   373.936  mm,
	W =    45.096 deg,	P =    12.591 deg,	R =   -22.909 deg
   GP2:
	UF : 0, UT : 1,
	J1=     0.000 deg,	J2=   180.000 deg
};
P[41]{
   GP1:
	UF : 1, UT : 1,		CONFIG : 'N U T, 0, 0, 0',
	X =  2134.406  mm,	Y =   435.630  mm,	Z =   299.420  mm,
	W =    43.046 deg,	P =    14.628 deg,	R =   -43.061 deg
   GP2:
	UF : 0, UT : 1,
	J1=     0.000 deg,	J2=   180.000 deg
};
P[42]{
   GP1:
	UF : 1, UT : 1,		CONFIG : 'N U T, 0, 0, 0',
	X =  2106.272  mm,	Y =   434.710  mm,	Z =   300.157  mm,
	W =    44.042 deg,	P =    10.806 deg,	R =   -14.045 deg
   GP2:
	UF : 0, UT : 1,
	J1=     0.000 deg,	J2=   180.000 deg
};
P[43]{
   GP1:
	UF : 1, UT : 1,		CONFIG : 'N U T, 0, 0, 0',
	X =  2097.132  mm,	Y =   436.405  mm,	Z =   293.176  mm,
	W =    47.286 deg,	P =    18.122 deg,	R =   -38.346 deg
   GP2:
	UF : 0, UT : 1,
	J1=     0.000 deg,	J2=   180.000 deg
};
P[44]{
   GP1:
	UF : 1, UT : 1,		CONFIG : 'N U T, 0, 0, 0',
	X =  2094.274  mm,	Y =   437.963  mm,	Z =   289.318  mm,
	W =    54.772 deg,	P =    18.651 deg,	R =   -46.003 deg
   GP2:
	UF : 0, UT : 1,
	J1=     0.000 deg,	J2=   180.000 deg
};
P[45]{
   GP1:
	UF : 1, UT : 1,		CONFIG : 'N U T, 0, 0, 0',
	X =  2119.797  mm,	Y =   296.237  mm,	Z =   373.936  mm,
	W =    45.096 deg,	P =    12.591 deg,	R =   -14.745 deg
   GP2:
	UF : 0, UT : 1,
	J1=     0.000 deg,	J2=   180.000 deg
};
P[46]{
   GP1:
	UF : 1, UT : 1,		CONFIG : 'N U T, 0, 0, 0',
	X =  2194.797  mm,	Y =   327.474  mm,	Z =   373.936  mm,
	W =    45.096 deg,	P =    12.591 deg,	R =   -14.745 deg
   GP2:
	UF : 0, UT : 1,
	J1=     0.000 deg,	J2=   180.000 deg
};
P[47]{
   GP1:
	UF : 1, UT : 1,		CONFIG : 'N U T, 0, 0, 0',
	X =  2190.044  mm,	Y =   437.665  mm,	Z =   298.404  mm,
	W =    43.151 deg,	P =    13.425 deg,	R =   -13.910 deg
   GP2:
	UF : 0, UT : 1,
	J1=     0.000 deg,	J2=   180.000 deg
};
P[48]{
   GP1:
	UF : 1, UT : 1,		CONFIG : 'N U T, 0, 0, 0',
	X =  2154.848  mm,	Y =   434.743  mm,	Z =   300.942  mm,
	W =    44.489 deg,	P =     7.391 deg,	R =    13.127 deg
   GP2:
	UF : 0, UT : 1,
	J1=     0.000 deg,	J2=   180.000 deg
};
P[49]{
   GP1:
	UF : 1, UT : 1,		CONFIG : 'N U T, 0, 0, 0',
	X =  2194.797  mm,	Y =   327.474  mm,	Z =   373.936  mm,
	W =    45.096 deg,	P =    12.591 deg,	R =   -14.745 deg
   GP2:
	UF : 0, UT : 1,
	J1=     0.000 deg,	J2=   180.000 deg
};
P[50]{
   GP1:
	UF : 1, UT : 1,		CONFIG : 'N U T, 0, 0, 0',
	X =  2194.797  mm,	Y =    65.474  mm,	Z =   373.936  mm,
	W =    45.096 deg,	P =    12.591 deg,	R =   -14.745 deg
   GP2:
	UF : 0, UT : 1,
	J1=     0.000 deg,	J2=   180.000 deg
};
P[51]{
   GP1:
	UF : 1, UT : 1,		CONFIG : 'N U T, 0, 0, 0',
	X =  2094.797  mm,	Y =   -75.526  mm,	Z =   373.936  mm,
	W =   -29.024 deg,	P =    38.011 deg,	R =    45.493 deg
   GP2:
	UF : 0, UT : 1,
	J1=     0.000 deg,	J2=   180.000 deg
};
P[52]{
   GP1:
	UF : 1, UT : 1,		CONFIG : 'N U T, 0, 0, 0',
	X =  2094.797  mm,	Y =  -377.526  mm,	Z =   373.936  mm,
	W =   -46.453 deg,	P =     -.249 deg,	R =    -2.725 deg
   GP2:
	UF : 0, UT : 1,
	J1=     0.000 deg,	J2=   180.000 deg
};
P[53]{
   GP1:
	UF : 1, UT : 1,		CONFIG : 'N U T, 0, 0, 0',
	X =  2134.347  mm,	Y =  -436.629  mm,	Z =   299.531  mm,
	W =   -44.975 deg,	P =    -1.475 deg,	R =    21.092 deg
   GP2:
	UF : 0, UT : 1,
	J1=      .000 deg,	J2=   180.000 deg
};
P[54]{
   GP1:
	UF : 1, UT : 1,		CONFIG : 'N U T, 0, 0, 0',
	X =  2104.548  mm,	Y =  -437.996  mm,	Z =   297.946  mm,
	W =   -44.604 deg,	P =     6.705 deg,	R =     6.752 deg
   GP2:
	UF : 0, UT : 1,
	J1=     0.000 deg,	J2=   180.000 deg
};
P[55]{
   GP1:
	UF : 1, UT : 1,		CONFIG : 'N U T, 0, 0, 0',
	X =  2096.858  mm,	Y =  -440.258  mm,	Z =   294.682  mm,
	W =   -41.574 deg,	P =     1.292 deg,	R =    11.594 deg
   GP2:
	UF : 0, UT : 1,
	J1=     0.000 deg,	J2=   180.000 deg
};
P[56]{
   GP1:
	UF : 1, UT : 1,		CONFIG : 'N U T, 0, 0, 0',
	X =  2091.823  mm,	Y =  -441.524  mm,	Z =   289.290  mm,
	W =   -42.365 deg,	P =    -7.029 deg,	R =    17.395 deg
   GP2:
	UF : 0, UT : 1,
	J1=     0.000 deg,	J2=   180.000 deg
};
P[57]{
   GP1:
	UF : 1, UT : 1,		CONFIG : 'N U T, 0, 0, 0',
	X =  2067.441  mm,	Y =  -278.531  mm,	Z =   454.279  mm,
	W =   -44.604 deg,	P =     6.705 deg,	R =    14.917 deg
   GP2:
	UF : 0, UT : 1,
	J1=     0.000 deg,	J2=   180.000 deg
};
P[58]{
   GP1:
	UF : 1, UT : 1,		CONFIG : 'N U T, 0, 0, 0',
	X =  2206.993  mm,	Y =  -383.344  mm,	Z =   379.133  mm,
	W =   -40.009 deg,	P =    25.912 deg,	R =    25.468 deg
   GP2:
	UF : 0, UT : 1,
	J1=     0.000 deg,	J2=   180.000 deg
};
P[59]{
   GP1:
	UF : 1, UT : 1,		CONFIG : 'N U T, 0, 0, 0',
	X =  2157.105  mm,	Y =  -437.897  mm,	Z =   300.163  mm,
	W =   -41.033 deg,	P =    20.379 deg,	R =     1.032 deg
   GP2:
	UF : 0, UT : 1,
	J1=     0.000 deg,	J2=   180.000 deg
};
P[60]{
   GP1:
	UF : 1, UT : 1,		CONFIG : 'N U T, 0, 0, 0',
	X =  2187.873  mm,	Y =  -436.002  mm,	Z =   298.148  mm,
	W =   -44.045 deg,	P =    10.291 deg,	R =    12.954 deg
   GP2:
	UF : 0, UT : 1,
	J1=     0.000 deg,	J2=   180.000 deg
};
P[61]{
   GP1:
	UF : 1, UT : 1,		CONFIG : 'N U T, 0, 0, 0',
	X =  2185.714  mm,	Y =  -325.864  mm,	Z =   402.368  mm,
	W =   -44.045 deg,	P =    10.291 deg,	R =    12.954 deg
   GP2:
	UF : 0, UT : 1,
	J1=     0.000 deg,	J2=   180.000 deg
};
P[62]{
   GP1:
	UF : 1, UT : 1,		CONFIG : 'N U T, 0, 0, 0',
	X =  1316.012  mm,	Y =   -61.784  mm,	Z =   400.825  mm,
	W =    11.867 deg,	P =    -6.405 deg,	R =   -40.983 deg
   GP2:
	UF : 0, UT : 1,
	J1=     0.000 deg,	J2=   180.000 deg
};
P[63]{
   GP1:
	UF : 1, UT : 1,		CONFIG : 'N U T, 0, 0, 0',
	X =  1323.445  mm,	Y =   -53.439  mm,	Z =   -20.480  mm,
	W =    24.441 deg,	P =    -8.933 deg,	R =   -71.136 deg
   GP2:
	UF : 0, UT : 1,
	J1=     0.000 deg,	J2=   180.000 deg
};
P[64]{
   GP1:
	UF : 1, UT : 1,		CONFIG : 'N U T, 0, 0, 0',
	X =  1338.138  mm,	Y =   -53.422  mm,	Z =   -39.866  mm,
	W =    27.066 deg,	P =    -9.807 deg,	R =   -71.565 deg
   GP2:
	UF : 0, UT : 1,
	J1=     0.000 deg,	J2=   180.000 deg
};
P[65]{
   GP1:
	UF : 1, UT : 1,		CONFIG : 'N U T, 0, 0, 0',
	X =  1337.981  mm,	Y =  -172.617  mm,	Z =   -42.986  mm,
	W =    30.946 deg,	P =    -7.916 deg,	R =   -82.479 deg
   GP2:
	UF : 0, UT : 1,
	J1=     0.000 deg,	J2=   180.000 deg
};
P[66]{
   GP1:
	UF : 1, UT : 1,		CONFIG : 'N U T, 0, 0, 0',
	X =  1338.658  mm,	Y =  -182.051  mm,	Z =   -41.273  mm,
	W =    27.609 deg,	P =   -16.706 deg,	R =   -92.220 deg
   GP2:
	UF : 0, UT : 1,
	J1=     0.000 deg,	J2=   180.000 deg
};
P[67]{
   GP1:
	UF : 1, UT : 1,		CONFIG : 'N U T, 0, 0, 0',
	X =  1305.014  mm,	Y =  -167.548  mm,	Z =    12.854  mm,
	W =    26.690 deg,	P =   -15.166 deg,	R =   -88.291 deg
   GP2:
	UF : 0, UT : 1,
	J1=     0.000 deg,	J2=   180.000 deg
};
P[68]{
   GP1:
	UF : 1, UT : 1,		CONFIG : 'N U T, 0, 0, 0',
	X =  1362.864  mm,	Y =  -149.434  mm,	Z =   300.607  mm,
	W =    16.584 deg,	P =   -24.331 deg,	R =   -52.652 deg
   GP2:
	UF : 0, UT : 1,
	J1=     0.000 deg,	J2=   180.000 deg
};
P[69]{
   GP1:
	UF : 1, UT : 1,		CONFIG : 'N U T, 0, 0, 0',
	X =  2075.191  mm,	Y =  -125.781  mm,	Z =  -461.526  mm,
	W =     1.303 deg,	P =    19.370 deg,	R =    -1.013 deg
   GP2:
	UF : 0, UT : 1,
	J1=    45.000 deg,	J2=   180.000 deg
};
P[70]{
   GP1:
	UF : 1, UT : 1,		CONFIG : 'N U T, 0, 0, 0',
	X =  2083.004  mm,	Y =   -55.853  mm,	Z =  -543.435  mm,
	W =     -.039 deg,	P =    29.544 deg,	R =     -.740 deg
   GP2:
	UF : 0, UT : 1,
	J1=    45.000 deg,	J2=   180.000 deg
};
P[71]{
   GP1:
	UF : 1, UT : 1,		CONFIG : 'N U T, 0, 0, 0',
	X =  2081.760  mm,	Y =  -183.846  mm,	Z =  -543.398  mm,
	W =     -.059 deg,	P =    29.545 deg,	R =     -.731 deg
   GP2:
	UF : 0, UT : 1,
	J1=    45.000 deg,	J2=   180.000 deg
};
P[72]{
   GP1:
	UF : 1, UT : 1,		CONFIG : 'N U T, 0, 0, 0',
	X =  2084.258  mm,	Y =  -164.318  mm,	Z =  -424.818  mm,
	W =     1.303 deg,	P =    19.370 deg,	R =    -1.013 deg
   GP2:
	UF : 0, UT : 1,
	J1=    45.000 deg,	J2=   180.000 deg
};
P[73]{
   GP1:
	UF : 1, UT : 1,		CONFIG : 'N U T, 0, 0, 0',
	X =  1032.407  mm,	Y =   -24.331  mm,	Z =   261.545  mm,
	W =     4.184 deg,	P =    27.142 deg,	R =     4.615 deg
   GP2:
	UF : 0, UT : 1,
	J1=    45.000 deg,	J2=   180.000 deg
};
P[74]{
   GP1:
	UF : 1, UT : 1,		CONFIG : 'N U B, 0, 0, 0',
	X =   353.784  mm,	Y =     3.997  mm,	Z =  2425.735  mm,
	W =     -.021 deg,	P =   -39.773 deg,	R =      .020 deg
   GP2:
	UF : 0, UT : 1,
	J1=    45.000 deg,	J2=   180.000 deg
};
P[75]{
   GP1:
	UF : 1, UT : 1,		CONFIG : 'N U T, 0, 0, 0',
	X =  1158.814  mm,	Y =  -274.490  mm,	Z =  1840.917  mm,
	W =   -10.829 deg,	P =   -15.923 deg,	R =    -3.213 deg
   GP2:
	UF : 0, UT : 1,
	J1=    90.000 deg,	J2=   135.000 deg
};
P[76]{
   GP1:
	UF : 1, UT : 1,		CONFIG : 'N U T, 0, 0, 0',
	X =  2194.335  mm,	Y =  -797.990  mm,	Z =   821.256  mm,
	W =   -12.714 deg,	P =     1.832 deg,	R =   -21.425 deg
   GP2:
	UF : 0, UT : 1,
	J1=    90.000 deg,	J2=   135.000 deg
};
P[77]{
   GP1:
	UF : 1, UT : 1,		CONFIG : 'N U T, 0, 0, 0',
	X =  2621.218  mm,	Y =  -912.348  mm,	Z =   659.568  mm,
	W =    -8.799 deg,	P =   -16.459 deg,	R =   -31.120 deg
   GP2:
	UF : 0, UT : 1,
	J1=    90.000 deg,	J2=   135.000 deg
};
P[78]{
   GP1:
	UF : 1, UT : 1,		CONFIG : 'N U T, 0, 0, 0',
	X =  2626.052  mm,	Y = -1029.575  mm,	Z =   488.976  mm,
	W =    -8.799 deg,	P =   -16.460 deg,	R =   -56.521 deg
   GP2:
	UF : 0, UT : 1,
	J1=    90.000 deg,	J2=   135.000 deg
};
P[79]{
   GP1:
	UF : 1, UT : 1,		CONFIG : 'N U T, 0, 0, 0',
	X =  2648.892  mm,	Y = -1044.870  mm,	Z =   442.100  mm,
	W =     -.413 deg,	P =    -3.555 deg,	R =   -57.986 deg
   GP2:
	UF : 0, UT : 1,
	J1=    90.000 deg,	J2=   135.000 deg
};
P[80]{
   GP1:
	UF : 1, UT : 1,		CONFIG : 'N U T, 0, 0, 0',
	X =  2674.605  mm,	Y = -1044.870  mm,	Z =   442.100  mm,
	W =     -.413 deg,	P =    -3.555 deg,	R =   -57.986 deg
   GP2:
	UF : 0, UT : 1,
	J1=    90.000 deg,	J2=   135.000 deg
};
P[81]{
   GP1:
	UF : 1, UT : 1,		CONFIG : 'N U T, 0, 0, 0',
	X =  2671.186  mm,	Y = -1007.991  mm,	Z =   499.177  mm,
	W =     6.649 deg,	P =   -10.542 deg,	R =   -58.667 deg
   GP2:
	UF : 0, UT : 1,
	J1=    90.000 deg,	J2=   135.000 deg
};
P[82]{
   GP1:
	UF : 1, UT : 1,		CONFIG : 'N U T, 0, 0, 0',
	X =  2671.115  mm,	Y =  -921.706  mm,	Z =   607.043  mm,
	W =     3.584 deg,	P =   -15.365 deg,	R =   -57.980 deg
   GP2:
	UF : 0, UT : 1,
	J1=    90.000 deg,	J2=   135.000 deg
};
P[83]{
   GP1:
	UF : 1, UT : 1,		CONFIG : 'N U T, 0, 0, 0',
	X =  2626.997  mm,	Y =  -751.318  mm,	Z =   885.579  mm,
	W =     5.894 deg,	P =   -21.990 deg,	R =   -35.568 deg
   GP2:
	UF : 0, UT : 1,
	J1=    90.000 deg,	J2=   135.000 deg
};
P[84]{
   GP1:
	UF : 1, UT : 1,		CONFIG : 'N U T, 0, 0, 0',
	X =  1599.653  mm,	Y =  -734.724  mm,	Z =  1199.941  mm,
	W =   -10.725 deg,	P =     6.521 deg,	R =    -7.813 deg
   GP2:
	UF : 0, UT : 1,
	J1=    90.000 deg,	J2=   135.000 deg
};
P[85]{
   GP1:
	UF : 1, UT : 1,		CONFIG : 'N U B, 0, 0, 0',
	X =   353.784  mm,	Y =     3.997  mm,	Z =  2425.735  mm,
	W =     -.021 deg,	P =   -39.773 deg,	R =      .020 deg
   GP2:
	UF : 0, UT : 1,
	J1=    90.000 deg,	J2=   135.000 deg
};
P[86]{
   GP1:
	UF : 1, UT : 1,
	J1=    33.588 deg,	J2=   -79.149 deg,	J3=    33.175 deg,
	J4=    61.799 deg,	J5=   -86.287 deg,	J6=     5.026 deg
   GP2:
	UF : 0, UT : 1,
	J1=   170.000 deg,	J2=     0.000 deg
};
P[87]{
   GP1:
	UF : 1, UT : 1,		CONFIG : 'N U T, 0, 0, 0',
	X =   930.680  mm,	Y =     3.607  mm,	Z =  1094.838  mm,
	W =   -52.090 deg,	P =    -5.757 deg,	R =     7.338 deg
   GP2:
	UF : 0, UT : 1,
	J1=   170.000 deg,	J2=     0.000 deg
};
P[88]{
   GP1:
	UF : 1, UT : 1,		CONFIG : 'N U T, 0, 0, 0',
	X =  1196.263  mm,	Y =  -372.062  mm,	Z =  1047.575  mm,
	W =   -43.308 deg,	P =   -32.848 deg,	R =   -32.628 deg
   GP2:
	UF : 0, UT : 1,
	J1=   170.000 deg,	J2=     0.000 deg
};
P[89]{
   GP1:
	UF : 1, UT : 1,		CONFIG : 'N U T, 0, 0, 0',
	X =  1207.072  mm,	Y =  -455.555  mm,	Z =  1039.706  mm,
	W =   -38.963 deg,	P =   -26.708 deg,	R =   -37.905 deg
   GP2:
	UF : 0, UT : 1,
	J1=   170.000 deg,	J2=     0.000 deg
};
P[90]{
   GP1:
	UF : 1, UT : 1,		CONFIG : 'N U T, 0, 0, 0',
	X =  1184.106  mm,	Y =  -512.068  mm,	Z =   986.287  mm,
	W =   -38.904 deg,	P =   -26.674 deg,	R =   -37.920 deg
   GP2:
	UF : 0, UT : 1,
	J1=   170.000 deg,	J2=      .000 deg
};
P[91]{
   GP1:
	UF : 1, UT : 1,		CONFIG : 'N U T, 0, 0, 0',
	X =  1299.178  mm,	Y =  -510.077  mm,	Z =   969.589  mm,
	W =   -31.410 deg,	P =   -32.305 deg,	R =   -41.743 deg
   GP2:
	UF : 0, UT : 1,
	J1=   170.000 deg,	J2=     0.000 deg
};
P[92]{
   GP1:
	UF : 1, UT : 1,		CONFIG : 'N U T, 0, 0, 0',
	X =  1304.520  mm,	Y =  -509.278  mm,	Z =   968.518  mm,
	W =   -31.410 deg,	P =   -32.305 deg,	R =   -29.949 deg
   GP2:
	UF : 0, UT : 1,
	J1=   170.000 deg,	J2=     0.000 deg
};
P[93]{
   GP1:
	UF : 1, UT : 1,		CONFIG : 'N U T, 0, 0, 0',
	X =  1295.522  mm,	Y =  -454.651  mm,	Z =  1026.440  mm,
	W =   -31.404 deg,	P =   -32.304 deg,	R =   -19.489 deg
   GP2:
	UF : 0, UT : 1,
	J1=   170.000 deg,	J2=     0.000 deg
};
P[94]{
   GP1:
	UF : 1, UT : 1,		CONFIG : 'N U T, 0, 0, 0',
	X =  1261.804  mm,	Y =  -244.256  mm,	Z =  1027.758  mm,
	W =   -22.133 deg,	P =   -20.172 deg,	R =    -9.613 deg
   GP2:
	UF : 0, UT : 1,
	J1=   170.000 deg,	J2=     0.000 deg
};
P[95]{
   GP1:
	UF : 1, UT : 1,		CONFIG : 'N U T, 0, 0, 0',
	X =   922.521  mm,	Y =    14.948  mm,	Z =  1180.907  mm,
	W =     4.751 deg,	P =    -2.174 deg,	R =    -1.174 deg
   GP2:
	UF : 0, UT : 1,
	J1=   170.000 deg,	J2=     0.000 deg
};
P[96]{
   GP1:
	UF : 1, UT : 1,		CONFIG : 'N U T, 0, 0, 0',
	X =  1022.000  mm,	Y =   102.282  mm,	Z =  1072.825  mm,
	W =    46.536 deg,	P =    -6.385 deg,	R =    -1.458 deg
   GP2:
	UF : 0, UT : 1,
	J1=   170.000 deg,	J2=     0.000 deg
};
P[97]{
   GP1:
	UF : 1, UT : 1,		CONFIG : 'N U T, 0, 0, 0',
	X =  1223.679  mm,	Y =   325.606  mm,	Z =  1022.839  mm,
	W =    44.741 deg,	P =   -16.673 deg,	R =    20.469 deg
   GP2:
	UF : 0, UT : 1,
	J1=   170.000 deg,	J2=     0.000 deg
};
P[98]{
   GP1:
	UF : 1, UT : 1,		CONFIG : 'N U T, 0, 0, 0',
	X =  1183.505  mm,	Y =   506.499  mm,	Z =   988.674  mm,
	W =    41.747 deg,	P =   -22.568 deg,	R =    30.362 deg
   GP2:
	UF : 0, UT : 1,
	J1=   170.000 deg,	J2=     0.000 deg
};
P[99]{
   GP1:
	UF : 1, UT : 1,		CONFIG : 'N U T, 0, 0, 0',
	X =  1294.200  mm,	Y =   504.899  mm,	Z =   971.327  mm,
	W =    41.747 deg,	P =   -22.568 deg,	R =    20.156 deg
   GP2:
	UF : 0, UT : 1,
	J1=   170.000 deg,	J2=     0.000 deg
};
P[100]{
   GP1:
	UF : 1, UT : 1,		CONFIG : 'N U T, 0, 0, 0',
	X =  1304.167  mm,	Y =   503.544  mm,	Z =   971.625  mm,
	W =    41.759 deg,	P =   -22.575 deg,	R =     -.824 deg
   GP2:
	UF : 0, UT : 1,
	J1=   170.000 deg,	J2=      .000 deg
};
P[101]{
   GP1:
	UF : 1, UT : 1,		CONFIG : 'N U T, 0, 0, 0',
	X =  1296.325  mm,	Y =   478.096  mm,	Z =  1014.718  mm,
	W =    49.103 deg,	P =   -22.303 deg,	R =    -3.634 deg
   GP2:
	UF : 0, UT : 1,
	J1=   170.000 deg,	J2=     0.000 deg
};
P[102]{
   GP1:
	UF : 1, UT : 1,		CONFIG : 'N U T, 0, 0, 0',
	X =   930.679  mm,	Y =     3.607  mm,	Z =  1094.839  mm,
	W =    46.788 deg,	P =    -6.408 deg,	R =    -6.777 deg
   GP2:
	UF : 0, UT : 1,
	J1=   170.000 deg,	J2=     0.000 deg
};
P[103]{
   GP1:
	UF : 1, UT : 1,		CONFIG : 'N U T, 0, 0, 0',
	X =   930.679  mm,	Y =     3.607  mm,	Z =  1816.839  mm,
	W =     -.163 deg,	P =    -9.317 deg,	R =      .025 deg
   GP2:
	UF : 0, UT : 1,
	J1=   145.000 deg,	J2=     0.000 deg
};
P[104]{
   GP1:
	UF : 1, UT : 1,		CONFIG : 'N U T, 0, 0, 0',
	X =  1445.680  mm,	Y =   567.607  mm,	Z =  1511.839  mm,
	W =     -.170 deg,	P =   -23.530 deg,	R =      .027 deg
   GP2:
	UF : 0, UT : 1,
	J1=   145.000 deg,	J2=     0.000 deg
};
P[105]{
   GP1:
	UF : 1, UT : 1,		CONFIG : 'N U T, 0, 0, 0',
	X =  1617.202  mm,	Y =   691.351  mm,	Z =  1394.804  mm,
	W =     -.170 deg,	P =   -23.530 deg,	R =      .027 deg
   GP2:
	UF : 0, UT : 1,
	J1=   145.000 deg,	J2=     0.000 deg
};
P[106]{
   GP1:
	UF : 1, UT : 1,		CONFIG : 'N U T, 0, 0, 0',
	X =  1638.526  mm,	Y =   682.552  mm,	Z =  1338.481  mm,
	W =     -.026 deg,	P =   -13.810 deg,	R =     -.098 deg
   GP2:
	UF : 0, UT : 1,
	J1=   145.000 deg,	J2=      .000 deg
};
P[107]{
   GP1:
	UF : 1, UT : 1,		CONFIG : 'N U T, 0, 0, 0',
	X =  1638.367  mm,	Y =   523.326  mm,	Z =  1336.599  mm,
	W =     -.126 deg,	P =   -13.859 deg,	R =     -.103 deg
   GP2:
	UF : 0, UT : 1,
	J1=   145.000 deg,	J2=      .000 deg
};
P[108]{
   GP1:
	UF : 1, UT : 1,		CONFIG : 'N U T, 0, 0, 0',
	X =  1636.393  mm,	Y =   512.206  mm,	Z =  1362.086  mm,
	W =     0.000 deg,	P =    -9.999 deg,	R =     0.000 deg
   GP2:
	UF : 0, UT : 1,
	J1=   145.000 deg,	J2=     0.000 deg
};
P[109]{
   GP1:
	UF : 1, UT : 1,		CONFIG : 'N U T, 0, 0, 0',
	X =  1636.312  mm,	Y =   496.857  mm,	Z =  1338.432  mm,
	W =      .202 deg,	P =   -10.242 deg,	R =     -.079 deg
   GP2:
	UF : 0, UT : 1,
	J1=   144.999 deg,	J2=      .000 deg
};
P[110]{
   GP1:
	UF : 1, UT : 1,		CONFIG : 'N U T, 0, 0, 0',
	X =  1637.379  mm,	Y =   470.985  mm,	Z =  1336.679  mm,
	W =      .173 deg,	P =   -10.188 deg,	R =     -.060 deg
   GP2:
	UF : 0, UT : 1,
	J1=   145.000 deg,	J2=      .000 deg
};
P[111]{
   GP1:
	UF : 1, UT : 1,		CONFIG : 'N U T, 0, 0, 0',
	X =  1586.518  mm,	Y =   509.816  mm,	Z =  1403.680  mm,
	W =     6.149 deg,	P =   -10.971 deg,	R =     8.557 deg
   GP2:
	UF : 0, UT : 1,
	J1=   145.000 deg,	J2=     0.000 deg
};
P[112]{
   GP1:
	UF : 1, UT : 1,		CONFIG : 'N U T, 0, 0, 0',
	X =  1586.518  mm,	Y =   412.011  mm,	Z =  1403.680  mm,
	W =     6.149 deg,	P =   -10.971 deg,	R =     8.557 deg
   GP2:
	UF : 0, UT : 1,
	J1=   145.000 deg,	J2=     0.000 deg
};
P[113]{
   GP1:
	UF : 1, UT : 1,		CONFIG : 'N U T, 0, 0, 0',
	X =  1613.222  mm,	Y =   422.510  mm,	Z =  1343.907  mm,
	W =     1.983 deg,	P =   -10.379 deg,	R =     8.603 deg
   GP2:
	UF : 0, UT : 1,
	J1=   145.000 deg,	J2=      .000 deg
};
P[114]{
   GP1:
	UF : 1, UT : 1,		CONFIG : 'N U T, 0, 0, 0',
	X =  1615.518  mm,	Y =  -427.276  mm,	Z =  1342.059  mm,
	W =     1.023 deg,	P =   -10.236 deg,	R =     8.658 deg
   GP2:
	UF : 0, UT : 1,
	J1=   145.000 deg,	J2=      .000 deg
};
P[115]{
   GP1:
	UF : 1, UT : 1,		CONFIG : 'N U T, 0, 0, 0',
	X =  1614.487  mm,	Y =  -414.217  mm,	Z =  1373.130  mm,
	W =    -1.488 deg,	P =    -9.890 deg,	R =     8.601 deg
   GP2:
	UF : 0, UT : 1,
	J1=   145.000 deg,	J2=     0.000 deg
};
P[116]{
   GP1:
	UF : 1, UT : 1,		CONFIG : 'N U T, 0, 0, 0',
	X =  1614.487  mm,	Y =  -485.217  mm,	Z =  1373.130  mm,
	W =    -1.488 deg,	P =    -9.890 deg,	R =     8.601 deg
   GP2:
	UF : 0, UT : 1,
	J1=   145.000 deg,	J2=     0.000 deg
};
P[117]{
   GP1:
	UF : 1, UT : 1,		CONFIG : 'N U T, 0, 0, 0',
	X =  1635.151  mm,	Y =  -476.391  mm,	Z =  1332.553  mm,
	W =    -1.488 deg,	P =    -9.890 deg,	R =     8.601 deg
   GP2:
	UF : 0, UT : 1,
	J1=   145.000 deg,	J2=     0.000 deg
};
P[118]{
   GP1:
	UF : 1, UT : 1,		CONFIG : 'N U T, 0, 0, 0',
	X =  1635.151  mm,	Y =  -505.534  mm,	Z =  1332.553  mm,
	W =    -1.488 deg,	P =    -9.890 deg,	R =     8.601 deg
   GP2:
	UF : 0, UT : 1,
	J1=   145.000 deg,	J2=     0.000 deg
};
P[119]{
   GP1:
	UF : 1, UT : 1,		CONFIG : 'N U T, 0, 0, 0',
	X =  1640.887  mm,	Y =  -485.217  mm,	Z =  1373.130  mm,
	W =    -1.488 deg,	P =    -9.889 deg,	R =     8.601 deg
   GP2:
	UF : 0, UT : 1,
	J1=   145.000 deg,	J2=     0.000 deg
};
P[120]{
   GP1:
	UF : 1, UT : 1,		CONFIG : 'N U T, 0, 0, 0',
	X =  1640.887  mm,	Y =  -536.817  mm,	Z =  1373.131  mm,
	W =    -1.488 deg,	P =    -9.889 deg,	R =     8.601 deg
   GP2:
	UF : 0, UT : 1,
	J1=   145.000 deg,	J2=     0.000 deg
};
P[121]{
   GP1:
	UF : 1, UT : 1,		CONFIG : 'N U T, 0, 0, 0',
	X =  1637.863  mm,	Y =  -518.699  mm,	Z =  1338.876  mm,
	W =    -1.478 deg,	P =    -9.889 deg,	R =     8.595 deg
   GP2:
	UF : 0, UT : 1,
	J1=   145.000 deg,	J2=      .000 deg
};
P[122]{
   GP1:
	UF : 1, UT : 1,		CONFIG : 'N U T, 0, 0, 0',
	X =  1638.691  mm,	Y =  -684.628  mm,	Z =  1339.948  mm,
	W =    -1.478 deg,	P =    -9.889 deg,	R =     8.595 deg
   GP2:
	UF : 0, UT : 1,
	J1=   145.000 deg,	J2=     0.000 deg
};
P[123]{
   GP1:
	UF : 1, UT : 1,		CONFIG : 'N U T, 0, 0, 0',
	X =  1596.746  mm,	Y =  -672.062  mm,	Z =  1470.175  mm,
	W =    -5.399 deg,	P =   -32.279 deg,	R =    10.036 deg
   GP2:
	UF : 0, UT : 1,
	J1=   145.000 deg,	J2=     0.000 deg
};
P[124]{
   GP1:
	UF : 1, UT : 1,		CONFIG : 'N U T, 0, 0, 0',
	X =  1245.795  mm,	Y =  -672.061  mm,	Z =  1470.175  mm,
	W =    -5.399 deg,	P =   -32.279 deg,	R =    10.036 deg
   GP2:
	UF : 0, UT : 1,
	J1=   145.000 deg,	J2=     0.000 deg
};
P[125]{
   GP1:
	UF : 1, UT : 1,		CONFIG : 'N U T, 0, 0, 0',
	X =  1035.165  mm,	Y =   -65.668  mm,	Z =  1132.208  mm,
	W =   -71.166 deg,	P =    14.285 deg,	R =    21.053 deg
   GP2:
	UF : 0, UT : 1,
	J1=   145.000 deg,	J2=     0.000 deg
};
P[126]{
   GP1:
	UF : 1, UT : 1,		CONFIG : 'N U T, 0, 0, 0',
	X =   705.308  mm,	Y =   628.212  mm,	Z =   613.128  mm,
	W =   -27.520 deg,	P =   -35.242 deg,	R =      .008 deg
   GP2:
	UF : 0, UT : 1,
	J1=   180.000 deg,	J2=    25.000 deg
};
P[127]{
   GP1:
	UF : 1, UT : 1,		CONFIG : 'N U T, 0, 0, 0',
	X =   823.942  mm,	Y =   433.727  mm,	Z =   902.693  mm,
	W =   -21.025 deg,	P =   -36.625 deg,	R =   -18.671 deg
   GP2:
	UF : 0, UT : 1,
	J1=   180.000 deg,	J2=    25.000 deg
};
P[128]{
   GP1:
	UF : 1, UT : 1,		CONFIG : 'N U T, 0, 0, 0',
	X =  1066.797  mm,	Y =   261.908  mm,	Z =   798.255  mm,
	W =   -30.186 deg,	P =   -35.006 deg,	R =   -19.606 deg
   GP2:
	UF : 0, UT : 1,
	J1=   180.000 deg,	J2=    25.000 deg
};
P[129]{
   GP1:
	UF : 1, UT : 1,		CONFIG : 'N U T, 0, 0, 0',
	X =  1202.450  mm,	Y =   329.449  mm,	Z =   801.269  mm,
	W =   -38.255 deg,	P =   -37.591 deg,	R =    24.434 deg
   GP2:
	UF : 0, UT : 1,
	J1=   180.000 deg,	J2=    25.000 deg
};
P[130]{
   GP1:
	UF : 1, UT : 1,		CONFIG : 'N U T, 0, 0, 0',
	X =  1140.326  mm,	Y =   318.744  mm,	Z =   819.048  mm,
	W =   -38.472 deg,	P =   -39.741 deg,	R =    23.618 deg
   GP2:
	UF : 0, UT : 1,
	J1=   180.000 deg,	J2=    25.000 deg
};
P[131]{
   GP1:
	UF : 1, UT : 1,		CONFIG : 'N U T, 0, 0, 0',
	X =   823.942  mm,	Y =   433.727  mm,	Z =   902.693  mm,
	W =   -21.025 deg,	P =   -36.625 deg,	R =   -18.671 deg
   GP2:
	UF : 0, UT : 1,
	J1=   180.000 deg,	J2=    25.000 deg
};
P[132]{
   GP1:
	UF : 1, UT : 1,		CONFIG : 'N U T, 0, 0, 0',
	X =   513.685  mm,	Y =   530.238  mm,	Z =  1690.590  mm,
	W =     9.276 deg,	P =   -38.124 deg,	R =    -9.504 deg
   GP2:
	UF : 0, UT : 1,
	J1=   180.000 deg,	J2=    25.000 deg
};
P[133]{
   GP1:
	UF : 1, UT : 1,		CONFIG : 'N U T, 0, 0, 0',
	X =   747.111  mm,	Y =  -550.972  mm,	Z =  1852.693  mm,
	W =   -21.025 deg,	P =   -36.625 deg,	R =    58.139 deg
   GP2:
	UF : 0, UT : 1,
	J1=   180.000 deg,	J2=   -25.000 deg
};
P[134]{
   GP1:
	UF : 1, UT : 1,		CONFIG : 'N U T, 0, 0, 0',
	X =   823.111  mm,	Y =  -474.039  mm,	Z =   844.692  mm,
	W =    29.770 deg,	P =   -48.142 deg,	R =     9.424 deg
   GP2:
	UF : 0, UT : 1,
	J1=   180.000 deg,	J2=   -25.000 deg
};
P[135]{
   GP1:
	UF : 1, UT : 1,		CONFIG : 'N U T, 0, 0, 0',
	X =  1000.111  mm,	Y =  -331.972  mm,	Z =   844.692  mm,
	W =    29.770 deg,	P =   -48.142 deg,	R =    14.585 deg
   GP2:
	UF : 0, UT : 1,
	J1=   180.000 deg,	J2=   -25.000 deg
};
P[136]{
   GP1:
	UF : 1, UT : 1,		CONFIG : 'N U T, 0, 0, 0',
	X =  1066.661  mm,	Y =  -270.706  mm,	Z =   801.500  mm,
	W =    28.148 deg,	P =   -36.678 deg,	R =    23.142 deg
   GP2:
	UF : 0, UT : 1,
	J1=   180.000 deg,	J2=   -25.000 deg
};
P[137]{
   GP1:
	UF : 1, UT : 1,		CONFIG : 'N U T, 0, 0, 0',
	X =  1200.620  mm,	Y =  -331.568  mm,	Z =   803.018  mm,
	W =    28.151 deg,	P =   -36.679 deg,	R =   -15.561 deg
   GP2:
	UF : 0, UT : 1,
	J1=   180.000 deg,	J2=   -25.000 deg
};
P[138]{
   GP1:
	UF : 1, UT : 1,		CONFIG : 'N U T, 0, 0, 0',
	X =  1000.111  mm,	Y =  -290.401  mm,	Z =   844.692  mm,
	W =    29.770 deg,	P =   -48.142 deg,	R =    14.585 deg
   GP2:
	UF : 0, UT : 1,
	J1=   180.000 deg,	J2=   -25.000 deg
};
P[139]{
   GP1:
	UF : 1, UT : 1,		CONFIG : 'N U T, 0, 0, 0',
	X =   753.111  mm,	Y =  -492.972  mm,	Z =   844.692  mm,
	W =    29.770 deg,	P =   -48.142 deg,	R =      .554 deg
   GP2:
	UF : 0, UT : 1,
	J1=   180.000 deg,	J2=   -25.000 deg
};
P[140]{
   GP1:
	UF : 1, UT : 1,		CONFIG : 'N U T, 0, 0, 0',
	X =   775.537  mm,	Y =  -786.141  mm,	Z =  1946.429  mm,
	W =   -25.333 deg,	P =   -46.944 deg,	R =    33.761 deg
   GP2:
	UF : 0, UT : 1,
	J1=   180.000 deg,	J2=   -25.000 deg
};
P[141]{
   GP1:
	UF : 1, UT : 1,		CONFIG : 'N U B, 0, 0, 0',
	X =   351.047  mm,	Y =     7.833  mm,	Z =  2455.305  mm,
	W =     -.021 deg,	P =   -39.773 deg,	R =      .020 deg
   GP2:
	UF : 0, UT : 1,
	J1=   180.000 deg,	J2=   -25.000 deg
};
P[142]{
   GP1:
	UF : 1, UT : 1,
	J1=      .000 deg,	J2=   -45.001 deg,	J3=    65.001 deg,
	J4=     -.002 deg,	J5=   -69.998 deg,	J6=     -.000 deg
   GP2:
	UF : 0, UT : 1,
	J1=     -.000 deg,	J2=   180.000 deg
};
P[143]{
   GP1:
	UF : 1, UT : 1,		CONFIG : 'N U T, 0, 0, 0',
	X =   869.467  mm,	Y =    18.934  mm,	Z =   587.034  mm,
	W =      .000 deg,	P =    46.047 deg,	R =   177.513 deg
   GP2:
	UF : 0, UT : 1,
	J1=     0.000 deg,	J2=   180.000 deg
};
P[144]{
   GP1:
	UF : 1, UT : 1,		CONFIG : 'N U T, 0, 0, 0',
	X =  1114.467  mm,	Y =   405.934  mm,	Z =   239.034  mm,
	W =      .000 deg,	P =    46.047 deg,	R =   177.513 deg
   GP2:
	UF : 0, UT : 1,
	J1=     0.000 deg,	J2=   180.000 deg
};
P[145]{
   GP1:
	UF : 1, UT : 1,		CONFIG : 'N U T, 0, 0, 0',
	X =  1206.924  mm,	Y =   427.021  mm,	Z =    57.080  mm,
	W =    -1.752 deg,	P =    44.972 deg,	R =   177.535 deg
   GP2:
	UF : 0, UT : 1,
	J1=      .000 deg,	J2=   180.000 deg
};
P[146]{
   GP1:
	UF : 1, UT : 1,		CONFIG : 'N U T, 0, 0, 1',
	X =  1206.140  mm,	Y =  -427.698  mm,	Z =    56.637  mm,
	W =    -2.069 deg,	P =    44.969 deg,	R =   177.081 deg
   GP2:
	UF : 0, UT : 1,
	J1=      .000 deg,	J2=   180.000 deg
};
P[147]{
   GP1:
	UF : 1, UT : 1,		CONFIG : 'N U T, 0, 0, 0',
	X =   923.454  mm,	Y =  -408.589  mm,	Z =   283.662  mm,
	W =      .000 deg,	P =    46.047 deg,	R =   177.059 deg
   GP2:
	UF : 0, UT : 1,
	J1=     0.000 deg,	J2=   180.000 deg
};
P[148]{
   GP1:
	UF : 1, UT : 1,		CONFIG : 'N U T, 0, 0, 0',
	X =  1130.453  mm,	Y =  -517.053  mm,	Z =   181.663  mm,
	W =     2.080 deg,	P =     1.084 deg,	R =    -2.041 deg
   GP2:
	UF : 0, UT : 1,
	J1=     0.000 deg,	J2=   180.000 deg
};
P[149]{
   GP1:
	UF : 1, UT : 1,		CONFIG : 'N U T, 0, 0, 0',
	X =  1102.943  mm,	Y =  -510.504  mm,	Z =    48.370  mm,
	W =    12.699 deg,	P =      .451 deg,	R =    -2.017 deg
   GP2:
	UF : 0, UT : 1,
	J1=      .000 deg,	J2=   180.000 deg
};
P[150]{
   GP1:
	UF : 1, UT : 1,		CONFIG : 'N U T, 0, 0, 0',
	X =  1202.266  mm,	Y =  -511.688  mm,	Z =    52.866  mm,
	W =    12.689 deg,	P =      .452 deg,	R =    -2.011 deg
   GP2:
	UF : 0, UT : 1,
	J1=     0.000 deg,	J2=   180.000 deg
};
P[151]{
   GP1:
	UF : 1, UT : 1,		CONFIG : 'N U T, 0, 0, 0',
	X =  1223.716  mm,	Y =  -511.573  mm,	Z =    53.134  mm,
	W =    13.354 deg,	P =   -18.278 deg,	R =    -2.108 deg
   GP2:
	UF : 0, UT : 1,
	J1=      .000 deg,	J2=   180.000 deg
};
P[152]{
   GP1:
	UF : 1, UT : 1,		CONFIG : 'N U T, 0, 0, 0',
	X =  1090.505  mm,	Y =  -517.053  mm,	Z =   181.663  mm,
	W =     2.080 deg,	P =     1.084 deg,	R =    -2.041 deg
   GP2:
	UF : 0, UT : 1,
	J1=     0.000 deg,	J2=   180.000 deg
};
P[153]{
   GP1:
	UF : 1, UT : 1,		CONFIG : 'N U T, 0, 0, 0',
	X =  1090.505  mm,	Y =   514.887  mm,	Z =   181.663  mm,
	W =     2.080 deg,	P =     1.084 deg,	R =    -2.041 deg
   GP2:
	UF : 0, UT : 1,
	J1=     0.000 deg,	J2=   180.000 deg
};
P[154]{
   GP1:
	UF : 1, UT : 1,		CONFIG : 'N U T, 0, 0, 0',
	X =  1106.481  mm,	Y =   519.927  mm,	Z =    49.181  mm,
	W =    -7.126 deg,	P =     -.205 deg,	R =    -2.067 deg
   GP2:
	UF : 0, UT : 1,
	J1=      .000 deg,	J2=   180.000 deg
};
P[155]{
   GP1:
	UF : 1, UT : 1,		CONFIG : 'N U T, 0, 0, 0',
	X =  1202.837  mm,	Y =   518.103  mm,	Z =    50.802  mm,
	W =   -11.587 deg,	P =     -.382 deg,	R =    -2.035 deg
   GP2:
	UF : 0, UT : 1,
	J1=      .000 deg,	J2=   180.000 deg
};
P[156]{
   GP1:
	UF : 1, UT : 1,		CONFIG : 'N U T, 0, 0, 0',
	X =  1224.743  mm,	Y =   517.964  mm,	Z =    50.717  mm,
	W =   -10.969 deg,	P =   -17.304 deg,	R =    -2.152 deg
   GP2:
	UF : 0, UT : 1,
	J1=      .000 deg,	J2=   180.000 deg
};
P[157]{
   GP1:
	UF : 1, UT : 1,		CONFIG : 'N U T, 0, 0, 0',
	X =  1087.212  mm,	Y =   520.313  mm,	Z =   176.360  mm,
	W =     2.582 deg,	P =   -12.004 deg,	R =    -2.085 deg
   GP2:
	UF : 0, UT : 1,
	J1=     0.000 deg,	J2=   180.000 deg
};
P[158]{
   GP1:
	UF : 1, UT : 1,		CONFIG : 'N U T, 0, 0, 0',
	X =   837.505  mm,	Y =   514.887  mm,	Z =   282.662  mm,
	W =      .000 deg,	P =    46.047 deg,	R =   177.059 deg
   GP2:
	UF : 0, UT : 1,
	J1=     0.000 deg,	J2=   180.000 deg
};
P[159]{
   GP1:
	UF : 1, UT : 1,		CONFIG : 'N U T, 0, 0, 0',
	X =  1173.408  mm,	Y =   683.888  mm,	Z =   198.662  mm,
	W =    34.780 deg,	P =    32.325 deg,	R =  -130.535 deg
   GP2:
	UF : 0, UT : 1,
	J1=     0.000 deg,	J2=   180.000 deg
};
P[160]{
   GP1:
	UF : 1, UT : 1,		CONFIG : 'N U T, 0, 0, 0',
	X =  1231.889  mm,	Y =   686.007  mm,	Z =    54.636  mm,
	W =    34.694 deg,	P =    32.328 deg,	R =  -130.608 deg
   GP2:
	UF : 0, UT : 1,
	J1=      .000 deg,	J2=   180.000 deg
};
P[161]{
   GP1:
	UF : 1, UT : 1,		CONFIG : 'N U T, 0, 0, 0',
	X =  1228.875  mm,	Y =   475.852  mm,	Z =    57.970  mm,
	W =    34.693 deg,	P =    32.344 deg,	R =  -130.608 deg
   GP2:
	UF : 0, UT : 1,
	J1=      .000 deg,	J2=   180.000 deg
};
P[162]{
   GP1:
	UF : 1, UT : 1,		CONFIG : 'N U T, 0, 0, 0',
	X =  1067.129  mm,	Y =   481.180  mm,	Z =   216.044  mm,
	W =    34.780 deg,	P =    32.324 deg,	R =  -130.534 deg
   GP2:
	UF : 0, UT : 1,
	J1=     0.000 deg,	J2=   180.000 deg
};
P[163]{
   GP1:
	UF : 1, UT : 1,		CONFIG : 'N U T, 0, 0, 1',
	X =   937.609  mm,	Y =  -628.912  mm,	Z =   407.224  mm,
	W =   -23.252 deg,	P =    40.938 deg,	R =   145.208 deg
   GP2:
	UF : 0, UT : 1,
	J1=     0.000 deg,	J2=   180.000 deg
};
P[164]{
   GP1:
	UF : 1, UT : 1,		CONFIG : 'N U T, 0, 0, 1',
	X =  1201.032  mm,	Y =  -681.912  mm,	Z =   158.223  mm,
	W =   -42.401 deg,	P =    19.964 deg,	R =   108.964 deg
   GP2:
	UF : 0, UT : 1,
	J1=     0.000 deg,	J2=   180.000 deg
};
P[165]{
   GP1:
	UF : 1, UT : 1,		CONFIG : 'N U T, 0, 0, 1',
	X =  1224.521  mm,	Y =  -687.891  mm,	Z =    57.774  mm,
	W =   -41.547 deg,	P =    19.139 deg,	R =   110.306 deg
   GP2:
	UF : 0, UT : 1,
	J1=      .000 deg,	J2=   180.000 deg
};
P[166]{
   GP1:
	UF : 1, UT : 1,		CONFIG : 'N U T, 0, 0, 1',
	X =  1225.852  mm,	Y =  -476.874  mm,	Z =    57.460  mm,
	W =   -41.533 deg,	P =    19.138 deg,	R =   110.296 deg
   GP2:
	UF : 0, UT : 1,
	J1=      .000 deg,	J2=   180.000 deg
};
P[167]{
   GP1:
	UF : 1, UT : 1,		CONFIG : 'N U T, 0, 0, 0',
	X =  1086.293  mm,	Y =  -468.046  mm,	Z =   256.961  mm,
	W =   -41.896 deg,	P =    19.479 deg,	R =   109.976 deg
   GP2:
	UF : 0, UT : 1,
	J1=     0.000 deg,	J2=   180.000 deg
};
P[168]{
   GP1:
	UF : 1, UT : 1,		CONFIG : 'N U T, 0, 0, 0',
	X =   896.023  mm,	Y =  -893.038  mm,	Z =   448.479  mm,
	W =    41.766 deg,	P =    21.483 deg,	R =   -23.558 deg
   GP2:
	UF : 0, UT : 1,
	J1=     0.000 deg,	J2=   180.000 deg
};
P[169]{
   GP1:
	UF : 1, UT : 1,		CONFIG : 'N U T, 0, 0, 0',
	X =   896.023  mm,	Y =  -525.038  mm,	Z =   448.479  mm,
	W =    41.767 deg,	P =    21.484 deg,	R =   -23.557 deg
   GP2:
	UF : 0, UT : 1,
	J1=     0.000 deg,	J2=   190.858 deg
};
P[170]{
   GP1:
	UF : 1, UT : 1,		CONFIG : 'N U T, 0, 0, 0',
	X =  1109.023  mm,	Y =  -598.037  mm,	Z =   219.479  mm,
	W =    41.765 deg,	P =    21.483 deg,	R =   -41.551 deg
   GP2:
	UF : 0, UT : 1,
	J1=     0.000 deg,	J2=   190.858 deg
};
P[171]{
   GP1:
	UF : 1, UT : 1,		CONFIG : 'N U T, 0, 0, 0',
	X =  1168.995  mm,	Y =  -554.545  mm,	Z =    56.898  mm,
	W =    38.815 deg,	P =    24.855 deg,	R =   -38.452 deg
   GP2:
	UF : 0, UT : 1,
	J1=      .000 deg,	J2=   190.858 deg
};
P[172]{
   GP1:
	UF : 1, UT : 1,		CONFIG : 'N U T, 0, 0, 0',
	X =  1442.387  mm,	Y =  -609.120  mm,	Z =    58.479  mm,
	W =    30.335 deg,	P =    15.583 deg,	R =   -43.439 deg
   GP2:
	UF : 0, UT : 1,
	J1=      .000 deg,	J2=   190.858 deg
};
P[173]{
   GP1:
	UF : 1, UT : 1,		CONFIG : 'N U T, 0, 0, 0',
	X =  1433.417  mm,	Y =  -682.761  mm,	Z =   191.796  mm,
	W =    22.166 deg,	P =     7.570 deg,	R =   -45.177 deg
   GP2:
	UF : 0, UT : 1,
	J1=     0.000 deg,	J2=   190.858 deg
};
P[174]{
   GP1:
	UF : 1, UT : 1,		CONFIG : 'N U T, 0, 0, 0',
	X =  1312.935  mm,	Y =  -662.070  mm,	Z =   295.434  mm,
	W =    23.681 deg,	P =     9.068 deg,	R =   -44.953 deg
   GP2:
	UF : 0, UT : 1,
	J1=     0.000 deg,	J2=   190.858 deg
};
P[175]{
   GP1:
	UF : 1, UT : 1,		CONFIG : 'N U T, 0, 0, 0',
	X =   693.417  mm,	Y =  -638.600  mm,	Z =   413.516  mm,
	W =    25.419 deg,	P =    10.774 deg,	R =   -44.658 deg
   GP2:
	UF : 0, UT : 1,
	J1=     0.000 deg,	J2=   190.858 deg
};
P[176]{
   GP1:
	UF : 1, UT : 1,		CONFIG : 'N U T, 0, 0, 0',
	X =   942.177  mm,	Y =   781.580  mm,	Z =   142.099  mm,
	W =   -34.550 deg,	P =    38.563 deg,	R =    42.094 deg
   GP2:
	UF : 0, UT : 1,
	J1=     0.000 deg,	J2=   180.000 deg
};
P[177]{
   GP1:
	UF : 1, UT : 1,		CONFIG : 'N U T, 0, 0, 0',
	X =  1291.176  mm,	Y =   799.653  mm,	Z =   164.696  mm,
	W =   -34.550 deg,	P =    38.563 deg,	R =    42.094 deg
   GP2:
	UF : 0, UT : 1,
	J1=     0.000 deg,	J2=   180.000 deg
};
P[178]{
   GP1:
	UF : 1, UT : 1,		CONFIG : 'N U T, 0, 0, 0',
	X =  1295.461  mm,	Y =   763.009  mm,	Z =    55.899  mm,
	W =   -30.106 deg,	P =    35.165 deg,	R =    44.796 deg
   GP2:
	UF : 0, UT : 1,
	J1=      .000 deg,	J2=   180.000 deg
};
P[179]{
   GP1:
	UF : 1, UT : 1,		CONFIG : 'N U T, 0, 0, 0',
	X =  1571.086  mm,	Y =   760.626  mm,	Z =    54.881  mm,
	W =   -45.053 deg,	P =    16.620 deg,	R =    41.357 deg
   GP2:
	UF : 0, UT : 1,
	J1=      .000 deg,	J2=   180.000 deg
};
P[180]{
   GP1:
	UF : 1, UT : 1,		CONFIG : 'N U T, 0, 0, 0',
	X =  1551.954  mm,	Y =   778.681  mm,	Z =   144.754  mm,
	W =   -49.546 deg,	P =    16.109 deg,	R =    43.352 deg
   GP2:
	UF : 0, UT : 1,
	J1=     0.000 deg,	J2=   180.000 deg
};
P[181]{
   GP1:
	UF : 1, UT : 1,		CONFIG : 'N U T, 0, 0, 0',
	X =   870.379  mm,	Y =   778.605  mm,	Z =   144.706  mm,
	W =   -44.038 deg,	P =    20.520 deg,	R =    47.848 deg
   GP2:
	UF : 0, UT : 1,
	J1=     0.000 deg,	J2=   180.000 deg
};
P[182]{
   GP1:
	UF : 1, UT : 1,		CONFIG : 'N U T, 0, 0, 0',
	X =   974.554  mm,	Y =   454.643  mm,	Z =   993.563  mm,
	W =   -33.816 deg,	P =    14.085 deg,	R =    17.851 deg
   GP2:
	UF : 0, UT : 1,
	J1=     0.000 deg,	J2=   180.000 deg
};
P[183]{
   GP1:
	UF : 1, UT : 1,		CONFIG : 'N U B, 0, 0, 0',
	X =   351.047  mm,	Y =     7.833  mm,	Z =  2455.305  mm,
	W =     -.021 deg,	P =   -39.773 deg,	R =      .020 deg
   GP2:
	UF : 0, UT : 1,
	J1=     0.000 deg,	J2=   180.000 deg
};
P[184]{
   GP1:
	UF : 1, UT : 1,
	J1=   -10.722 deg,	J2=   -74.333 deg,	J3=    51.477 deg,
	J4=    -3.440 deg,	J5=  -105.888 deg,	J6=   152.481 deg
   GP2:
	UF : 0, UT : 1,
	J1=   180.000 deg,	J2=   180.000 deg
};
P[185]{
   GP1:
	UF : 1, UT : 1,		CONFIG : 'N U T, 0, 0, 0',
	X =   588.577  mm,	Y =   298.999  mm,	Z =   876.681  mm,
	W =   -18.946 deg,	P =    44.582 deg,	R =   168.812 deg
   GP2:
	UF : 0, UT : 1,
	J1=   180.000 deg,	J2=   180.000 deg
};
P[186]{
   GP1:
	UF : 1, UT : 1,		CONFIG : 'N U T, 0, 0, 0',
	X =   688.932  mm,	Y =   314.970  mm,	Z =   764.761  mm,
	W =   -18.743 deg,	P =    41.455 deg,	R =   154.013 deg
   GP2:
	UF : 0, UT : 1,
	J1=   180.000 deg,	J2=   180.000 deg
};
P[187]{
   GP1:
	UF : 1, UT : 1,		CONFIG : 'N U T, 0, 0, 0',
	X =   686.972  mm,	Y =   381.813  mm,	Z =   767.487  mm,
	W =   -33.672 deg,	P =    31.165 deg,	R =   147.999 deg
   GP2:
	UF : 0, UT : 1,
	J1=   179.999 deg,	J2=   180.000 deg
};
P[188]{
   GP1:
	UF : 1, UT : 1,		CONFIG : 'N U T, 0, 0, 0',
	X =   571.859  mm,	Y =   355.407  mm,	Z =   890.190  mm,
	W =   -40.409 deg,	P =    21.774 deg,	R =   135.318 deg
   GP2:
	UF : 0, UT : 1,
	J1=   180.000 deg,	J2=   180.000 deg
};
P[189]{
   GP1:
	UF : 1, UT : 1,		CONFIG : 'N U T, 0, 0, 0',
	X =   642.859  mm,	Y =   281.847  mm,	Z =   890.189  mm,
	W =   -40.407 deg,	P =    21.774 deg,	R =   118.081 deg
   GP2:
	UF : 0, UT : 1,
	J1=   180.000 deg,	J2=   180.000 deg
};
P[190]{
   GP1:
	UF : 1, UT : 1,		CONFIG : 'N U T, 0, 0, 0',
	X =   688.982  mm,	Y =   282.012  mm,	Z =   764.727  mm,
	W =   -39.531 deg,	P =    23.501 deg,	R =   116.498 deg
   GP2:
	UF : 0, UT : 1,
	J1=   180.000 deg,	J2=   180.000 deg
};
P[191]{
   GP1:
	UF : 1, UT : 1,		CONFIG : 'N U T, 0, 0, 1',
	X =   687.735  mm,	Y =  -277.604  mm,	Z =   765.790  mm,
	W =    42.217 deg,	P =    17.331 deg,	R =  -106.993 deg
   GP2:
	UF : 0, UT : 1,
	J1=   180.000 deg,	J2=   180.000 deg
};
P[192]{
   GP1:
	UF : 1, UT : 1,		CONFIG : 'N U T, 0, 0, 1',
	X =   660.939  mm,	Y =  -331.949  mm,	Z =   794.701  mm,
	W =    42.404 deg,	P =    16.748 deg,	R =  -107.282 deg
   GP2:
	UF : 0, UT : 1,
	J1=   180.000 deg,	J2=   180.000 deg
};
P[193]{
   GP1:
	UF : 1, UT : 1,		CONFIG : 'N U T, 0, 0, 0',
	X =  2780.753  mm,	Y =    85.443  mm,	Z =   844.936  mm,
	W =   -24.896 deg,	P =    26.710 deg,	R =    44.095 deg
   GP2:
	UF : 0, UT : 1,
	J1=    90.000 deg,	J2=   180.000 deg
};
P[194]{
   GP1:
	UF : 1, UT : 1,		CONFIG : 'N U T, 0, 0, 1',
	X =   686.395  mm,	Y =  -319.415  mm,	Z =   767.232  mm,
	W =    42.396 deg,	P =    16.802 deg,	R =  -107.252 deg
   GP2:
	UF : 0, UT : 1,
	J1=   180.000 deg,	J2=   180.000 deg
};
P[195]{
   GP1:
	UF : 1, UT : 1,		CONFIG : 'N U T, 0, 0, 1',
	X =   686.344  mm,	Y =  -395.538  mm,	Z =   767.374  mm,
	W =    42.332 deg,	P =    16.923 deg,	R =  -127.294 deg
   GP2:
	UF : 0, UT : 1,
	J1=   180.000 deg,	J2=   180.000 deg
};
P[196]{
   GP1:
	UF : 1, UT : 1,		CONFIG : 'N U T, 0, 0, 1',
	X =   399.609  mm,	Y =  -296.816  mm,	Z =  1066.129  mm,
	W =    41.082 deg,	P =    20.266 deg,	R =  -127.997 deg
   GP2:
	UF : 0, UT : 1,
	J1=   180.000 deg,	J2=   180.000 deg
};
P[197]{
   GP1:
	UF : 1, UT : 1,
	J1=   -50.020 deg,	J2=   -69.917 deg,	J3=    26.974 deg,
	J4=   -21.929 deg,	J5=   -51.874 deg,	J6=    85.098 deg
   GP2:
	UF : 0, UT : 1,
	J1=   180.000 deg,	J2=   196.129 deg
};
P[198]{
   GP1:
	UF : 1, UT : 1,		CONFIG : 'N U T, 0, 0, 0',
	X =   901.665  mm,	Y =  -745.253  mm,	Z =  1087.372  mm,
	W =   -38.429 deg,	P =   -34.649 deg,	R =      .780 deg
   GP2:
	UF : 0, UT : 1,
	J1=   180.000 deg,	J2=   196.129 deg
};
P[199]{
   GP1:
	UF : 1, UT : 1,		CONFIG : 'N U T, 0, 0, 0',
	X =   933.220  mm,	Y =  -797.225  mm,	Z =  1036.983  mm,
	W =   -35.805 deg,	P =   -29.184 deg,	R =    -4.130 deg
   GP2:
	UF : 0, UT : 1,
	J1=   180.000 deg,	J2=   196.129 deg
};
P[200]{
   GP1:
	UF : 1, UT : 1,		CONFIG : 'N U T, 0, 0, 0',
	X =  1028.274  mm,	Y =  -768.347  mm,	Z =  1035.766  mm,
	W =   -48.186 deg,	P =   -30.992 deg,	R =     6.378 deg
   GP2:
	UF : 0, UT : 1,
	J1=   180.000 deg,	J2=   196.129 deg
};
P[201]{
   GP1:
	UF : 1, UT : 1,		CONFIG : 'N U T, 0, 0, 0',
	X =  1003.246  mm,	Y =  -747.467  mm,	Z =  1073.858  mm,
	W =   -73.601 deg,	P =   -18.162 deg,	R =    24.579 deg
   GP2:
	UF : 0, UT : 1,
	J1=   180.000 deg,	J2=   196.129 deg
};
P[202]{
   GP1:
	UF : 1, UT : 1,		CONFIG : 'N U T, 0, 0, 0',
	X =   635.246  mm,	Y =  -747.467  mm,	Z =  1080.599  mm,
	W =   -73.601 deg,	P =   -18.162 deg,	R =    24.579 deg
   GP2:
	UF : 0, UT : 1,
	J1=   180.000 deg,	J2=   196.129 deg
};
P[203]{
   GP1:
	UF : 1, UT : 1,		CONFIG : 'N U T, 0, 0, 0',
	X =   863.342  mm,	Y =  -725.478  mm,	Z =  1030.928  mm,
	W =     -.609 deg,	P =   -11.317 deg,	R =    19.232 deg
   GP2:
	UF : 0, UT : 1,
	J1=   180.000 deg,	J2=   196.129 deg
};
P[204]{
   GP1:
	UF : 1, UT : 1,		CONFIG : 'N U T, 0, 0, 0',
	X =   882.351  mm,	Y =  -732.230  mm,	Z =   976.636  mm,
	W =     -.603 deg,	P =   -11.312 deg,	R =    19.225 deg
   GP2:
	UF : 0, UT : 1,
	J1=   180.000 deg,	J2=   196.129 deg
};
P[205]{
   GP1:
	UF : 1, UT : 1,		CONFIG : 'N U T, 0, 0, 0',
	X =   897.394  mm,	Y =  -786.978  mm,	Z =   978.292  mm,
	W =      .775 deg,	P =    -4.353 deg,	R =    18.091 deg
   GP2:
	UF : 0, UT : 1,
	J1=   180.000 deg,	J2=   196.129 deg
};
P[206]{
   GP1:
	UF : 1, UT : 1,		CONFIG : 'N U T, 0, 0, 0',
	X =   891.737  mm,	Y =  -780.782  mm,	Z =  1041.865  mm,
	W =     -.266 deg,	P =   -10.779 deg,	R =    18.391 deg
   GP2:
	UF : 0, UT : 1,
	J1=   180.000 deg,	J2=   196.129 deg
};
P[207]{
   GP1:
	UF : 1, UT : 1,		CONFIG : 'N U T, 0, 0, 0',
	X =   439.173  mm,	Y =  -215.827  mm,	Z =  1826.127  mm,
	W =  -100.113 deg,	P =   -16.084 deg,	R =    32.515 deg
   GP2:
	UF : 0, UT : 1,
	J1=   180.000 deg,	J2=   196.129 deg
};
P[208]{
   GP1:
	UF : 1, UT : 1,		CONFIG : 'N U T, 0, 0, 0',
	X =   417.228  mm,	Y =   731.748  mm,	Z =  1722.425  mm,
	W =    31.808 deg,	P =   -58.935 deg,	R =    27.008 deg
   GP2:
	UF : 0, UT : 1,
	J1=   180.000 deg,	J2=   162.834 deg
};
P[209]{
   GP1:
	UF : 1, UT : 1,		CONFIG : 'N U T, 0, 0, 0',
	X =   892.925  mm,	Y =   804.354  mm,	Z =  1049.649  mm,
	W =    26.626 deg,	P =   -37.722 deg,	R =    33.504 deg
   GP2:
	UF : 0, UT : 1,
	J1=   180.000 deg,	J2=   162.834 deg
};
P[210]{
   GP1:
	UF : 1, UT : 1,		CONFIG : 'N U T, 0, 0, 0',
	X =   945.035  mm,	Y =   821.604  mm,	Z =  1034.094  mm,
	W =    26.239 deg,	P =   -37.738 deg,	R =    26.839 deg
   GP2:
	UF : 0, UT : 1,
	J1=   179.999 deg,	J2=   162.834 deg
};
P[211]{
   GP1:
	UF : 1, UT : 1,		CONFIG : 'N U T, 0, 0, 0',
	X =  1040.438  mm,	Y =   789.359  mm,	Z =  1035.196  mm,
	W =    34.470 deg,	P =   -41.842 deg,	R =    17.130 deg
   GP2:
	UF : 0, UT : 1,
	J1=   179.999 deg,	J2=   162.834 deg
};
P[212]{
   GP1:
	UF : 1, UT : 1,		CONFIG : 'N U T, 0, 0, 0',
	X =  1023.433  mm,	Y =   777.172  mm,	Z =  1060.439  mm,
	W =    35.127 deg,	P =   -46.999 deg,	R =     8.144 deg
   GP2:
	UF : 0, UT : 1,
	J1=   180.000 deg,	J2=   162.834 deg
};
P[213]{
   GP1:
	UF : 1, UT : 1,		CONFIG : 'N U T, 0, 0, 0',
	X =   647.433  mm,	Y =   777.171  mm,	Z =  1087.913  mm,
	W =    35.127 deg,	P =   -46.999 deg,	R =     8.144 deg
   GP2:
	UF : 0, UT : 1,
	J1=   180.000 deg,	J2=   162.834 deg
};
P[214]{
   GP1:
	UF : 1, UT : 1,		CONFIG : 'N U T, 0, 0, 0',
	X =   875.269  mm,	Y =   770.680  mm,	Z =  1039.359  mm,
	W =    -7.923 deg,	P =    -8.129 deg,	R =    27.445 deg
   GP2:
